(* CODESYS project festo_motion_fhpp_3.library
   Company: Festo AG & Co. KG
   DefaultNamespace: FML
   Title: Festo_Motion_FHPP_3
   Description: Library to control and parameterise drives from Festo with FHPP
   Author: chmm
   Version: 3.5.7.21

Project tree, tasks and I/O mapping:
  libraries: Standard, * (System)
  Enums/
    data type E_FML_DIAG_EVENT
    data type E_FML_FPC_MODUS
    data type E_FML_FPC_REQ_ID
    data type E_FML_FPC_RESP_ID
    data type E_FML_OPM
    data type E_FML_DEVICE_TYPE
    data type E_FML_FPC_STATUS_CATEGORY
    data type E_FML_FPC_STATUS_ID_FUNCTION_BLOCK
    data type E_FML_FPC_STATUS_ID_FILE_TRANSFER
  Internal/
    Blocks/
      ReadWriteData/
        function block FHPP_PLUS_Read [ST]
        function block FPC_Write [ST]
        function block FHPP_Read [ST]
        function block FHPP_PLUS_Write [ST]
        function block FHPP_Write [ST]
        function block FPC_Read [ST]
      FaultString/
        function ErrorList_CMMP_AS [ST]
        function ErrorList_CMMD_CMMS [ST]
        function ErrorList_CMMO_ST_EMCA_EC [ST]
        function FaultString [ST]
        function ErrorList_SFC_MTR [ST]
      function GetStatusMessage [ST]
      function GetStateOPMString [ST]
      function FML_DiagEventString [ST]
      function FML_TimeStamp [ST]
      function FormatInt [ST]
      function GetOPMString [ST]
    Enums/
      data type FML_FPC_FILE_TRANSFER_CONTROL
    Structs/
      FPC/
        data type DT_FPC
        data type DT_FPC_DATA
      FHPP/
        data type DT_CCON
        data type DT_CPOS
        data type DT_SCON
        data type DT_FHPP_DATA_IN
        data type DT_SPOS
        data type DT_FHPP
        data type DT_FHPP_DATA_OUT
      FHPP_PLUS/
        data type DT_FHPP_PLUS_OBJECT
        data type DT_FHPP_PLUS
      data type UCHAR
  Structs/
    data type DT_FML_REF
    data type DT_FML_PRM_DESCRIPTION
    data type DT_FML_PRM_DIAGMESSAGE
    data type DT_FML_DiagTable
    data type DT_FML_STATUS
    data type DT_FML_FPC_FILE_TRANSFER
  VISU/
    visualisation VIS_FPC_PNU
    visualisation VIS_FPC_DIAG_BUFFER
    visualisation VIS_FPC_DIRMP
    visualisation VIS_FPC_DATA_OBJECT
    visualisation VIS_FHPP_CTRL
    visualisation VIS_FPC_DIAG
    visualisation VIS_FPC_MULTI
    visualisation VIS_FPC_FILE_ARRAY
  Blocks/
    function block FHPP_CTRL [ST]
    function block FML_Read [ST]
    function block FML_Write [ST]
    Parameterize/
      function block FPC_DIAG_BUFFER [ST]
      function block FPC_MULTI [ST]
      function block FPC_PNU [ST]
      function block FPC_DATA_OBJECT [ST]
      function block FPC_DIAG [ST]
      function block FPC_FILE_ARRAY [ST]: CalculateFilesize, NextSequence
      function block FPC_DIRMP [ST]
  text list GlobalTextList
*)

// Structs/DT_FML_REF
(* ============================================================================
   FESTO AG & Co. KG, Esslingen - Copyright 2013. All rights reserved.                       
 ---------------------------------------------------------------------
 Data Type:     DT_FML_REF  
 Description:   data structure for Parametertransmission
 Version:       V3.1        
 Composer:      bejk
 Last Update:   26.06.2014                                                                           
 ---------------------------------------------------------------------
DATE        Name              	Activity                                                                              
11.03.2009  Benjamin Kilgus   	V1.0: created
13.05.2013  Rudolf Schenke    	V3.0: Formatting only
01.04.2014	Benjamin Kilgus	  	V3.1: extended to funktionality of EFPC
26.06.2014	Benjamin Kilgus	  	V3.1: extended FPCC_Packet/ FPCS_Packet
22.06.2015	Christian Hammer	adaptation to use this FB for all drives
08.09.2015	Christian Hammer	deleted 'ErrStr' with Error information
============================================================================ *)

TYPE DT_FML_REF :
	STRUCT
		(*data*)
		FHPP				: DT_FHPP;					// FHPP data
		FPC					: DT_FPC;					// FPC data
		FHPP_PLUS			: DT_FHPP_PLUS;				// FHPP+ data
	
		(*adjustments*)
		Modbus				: BOOL;						// Modbus is using
		HighByteFirst		: BOOL;						// Byteorder
		FPC_active			: BOOL;						// ParameterChannel (FPC) in use
	  	DeviceType			: E_FML_DEVICE_TYPE;		// Type of the Controller
		
		(*component infos*)
		MemberID	    	: INT:= 0;					// Current Member-ID
	 	MemberIDmax			: INT:= 0; 					// Maximum Member-ID
	  	Done          		: BOOL;     				// Execution Done 
	  	Err           		: BOOL;     				// Fault occured   
		
		(*request*)
		PNU           		: INT;	     				// Number of the Parameter 
	  	Subindex      		: DINT;    					// Subindex of the Parameter to Exchange 
		Value  				: DINT;     				// Value of the Parameter to Exchange
		DatatypeWR      	: USINT;    				// Length of the Parameter to Exchange in Byte
		ReqID				: E_FML_FPC_REQ_ID;
		FPCC_Packet			: DT_FML_FPC_FILE_TRANSFER; // File Transfer Packet Control
		FPCC_Modus			: DINT; 	  				// modus of parameter channel control

		(*response*)
		ActPNU        		: INT;	     				// Actual Number of the Parameter
	  	ActSubindex   		: DINT;    					// Actual Subindex of the Parameter 
	  	ActValue  			: DINT;     				// Read Value of Parameter
		DatatypeRD      	: USINT;    				// Actual Length of the Parameter in Byte
	  	RespID				: E_FML_FPC_RESP_ID;
	  	FPCS_Packet			: DT_FML_FPC_FILE_TRANSFER; // File Transfer Packet Status
		FPCS_Modus			: DINT; 	  				// modus of parameter channel status 
  END_STRUCT
END_TYPE

// Structs/DT_FML_PRM_DESCRIPTION
(* ============================================================================
   FESTO AG & Co. KG, Esslingen - Copyright (c) 2015. All rights reserved.                                   								
  -----------------------------------------------------------------------------  
 Description:    data structure for discription of the parameter   
 Last Update:    25.06.2014                                                                           
 ------------------------------------------------------------------------------
 Date        Name              	Activity                                                                              
 25.06.2014	 Benjamin Kilgus	created
 
 ============================================================================ *)

TYPE DT_FML_PRM_DESCRIPTION :
  STRUCT
	  PNU      	: INT ;		(* parameter number *)
	  SUBINDEX 	: INT ;		(* subindex of parameter *)
	  ACCESS   	: INT ;		(* 0 = read parameter / 1 = write parameter*)
	  VALUE    	: DINT ;	(* parameter value*)
	  Length	: USINT;	(* length of the parameter to exchange in byte (only necessary for SFC-DC and MTR-DCI) *)
  END_STRUCT
END_TYPE

// Structs/DT_FML_PRM_DIAGMESSAGE
(* ============================================================================
   FESTO AG & Co. KG, Esslingen - Copyright (c) 2015. All rights reserved.                                   								
  -----------------------------------------------------------------------------  
 Description:    data structure for diagnosis message   
 Last Update:    25.06.2014                                                                           
 ------------------------------------------------------------------------------
 Date        Name              	Activity                                                                              
 25.06.2014	 Benjamin Kilgus	created
 ============================================================================ *)

TYPE DT_FML_PRM_DIAGMESSAGE :
  STRUCT
	  DiagEvent          :E_FML_DIAG_EVENT;   	// event of message PNU 200/ PNU 210
	  DiagMsgNumber      :DINT;   			 	// message number PNU 201/ PNU 211
	  DiagTimeStamp      :DWORD;  				// time stamp of message PNU 202/ PNU 212
	  DiagMsgDescription :STRING; 				// description of message
  END_STRUCT
END_TYPE

// Enums/E_FML_DIAG_EVENT
(* ============================================================================
   FESTO AG & Co. KG, Esslingen - Copyright (c) 2015. All rights reserved.                                   								
  -----------------------------------------------------------------------------  
 Description:    enumeration for FML diagnosis event of the motorcontroller  
 Last Update:    22.06.2015                                                                           
 ------------------------------------------------------------------------------
 Date        Name                Activity                                                                              
 08.04.2014  Benjamin Kilgus	 created	 
 ============================================================================ *)

TYPE E_FML_DIAG_EVENT :
(
	none 				:= 0,
	error_comes     	:= 1,
	error_gone			:= 2,
	error_quit			:= 3,
	overflow_timestamp	:= 4,
	warning_comes		:= 5,
	warning_gone		:= 6,
	start_up_event  	:= 7,
	configuration		:= 8,
	information			:= 9
)INT;
END_TYPE

// Enums/E_FML_FPC_MODUS
(* ============================================================================
   FESTO AG & Co. KG, Esslingen - Copyright (c) 2015. All rights reserved.                                   								
  -----------------------------------------------------------------------------  
 Description:    enumeration for FML FPC Modus   
 Last Update:    25.06.2014                                                                           
 ------------------------------------------------------------------------------
 Date        Name              	Activity                                                                              
 01.04.2014  Benjamin Kilgus   	created 
 25.06.2014	Benjamin Kilgus	   	Type 4 and 5 added
 ============================================================================ *)

TYPE E_FML_FPC_MODUS :
(
	FML_FPC_MODUS_PNU_11BIT 	    := 0,	// transmit PNU 11 bit
	FML_FPC_MODUS_PNU_16BIT	 	    := 1,	// transmit PNU 16 bit
	FML_FPC_MODUS_DATA_OBJECT		:= 2,	// transmit internal data object
	FML_FPC_MODUS_CAN				:= 3,	// transmit CAN object
	FML_FPC_MODUS_ParameterFile	  	:= 4,	// transmit parameter file
	FML_FPC_MODUS_FirmwareUpdate  	:= 5	// transmit firmware file
)INT;
END_TYPE

// Enums/E_FML_FPC_REQ_ID
(* ============================================================================
   FESTO AG & Co. KG, Esslingen - Copyright (c) 2015. All rights reserved.                                   								
  -----------------------------------------------------------------------------  
 Description:    enumeration for FML FPC Modus   
 Last Update:    25.06.2014                                                                           
 ------------------------------------------------------------------------------
 Date        Name                Activity                                                                              
 25.06.2014	Benjamin Kilgus		 created
 ============================================================================ *)

TYPE E_FML_FPC_REQ_ID :
(
	FML_FPC_REQ_none	 			:= 0,	
	FML_FPC_REQ_read		 		:= 1,	
	FML_FPC_REQ_write_word			:= 2,	
	FML_FPC_REQ_write_dword			:= 3,	
	FML_FPC_REQ_read_file			:= 4,	
	FML_FPC_REQ_write_file			:= 5,
	FML_FPC_REQ_read_array			:= 6,
	FML_FPC_REQ_write_array_word	:= 7,
	FML_FPC_REQ_write_array_dword	:= 8,
	FML_FPC_REQ_read_array_elements	:= 9,
	FML_FPC_REQ_reseved0			:= 10,
	FML_FPC_REQ_write_byte			:= 11,
	FML_FPC_REQ_write_array_byte	:= 12,
	FML_FPC_REQ_read_lower_limit	:= 13,
	FML_FPC_REQ_read_upper_limit	:= 14	
)INT;
END_TYPE

// Enums/E_FML_FPC_RESP_ID
(* ============================================================================
   FESTO AG & Co. KG, Esslingen - Copyright (c) 2015. All rights reserved.                                   								
  -----------------------------------------------------------------------------  
 Description:    enumeration for FML FPC Modus   
 Last Update:    25.06.2014                                                                           
 ------------------------------------------------------------------------------
 Date        Name                Activity                                                                              
 25.06.2014	Benjamin Kilgus		 created
 ============================================================================ *)

TYPE E_FML_FPC_RESP_ID :
(
	FML_FPC_RESP_none	 				:= 0,	
	FML_FPC_RESP_word_done	 			:= 1,	
	FML_FPC_RESP_dword_done				:= 2,	
	FML_FPC_RESP_file_done				:= 3,	
	FML_FPC_RESP_word_array_done		:= 4,	
	FML_FPC_RESP_dword_array_done		:= 5,
	FML_FPC_RESP_error					:= 7,
	FML_FPC_RESP_read_array_elements	:= 9,
	FML_FPC_RESP_reseved0				:= 10,
	FML_FPC_RESP_byte_done				:= 11,
	FML_FPC_RESP_byte_array_done		:= 12		
)INT;
END_TYPE

// Enums/E_FML_OPM
(* ============================================================================
   FESTO AG & Co. KG, Esslingen - Copyright (c) 2015. All rights reserved.                                   								
  -----------------------------------------------------------------------------  
 Description:    enumeration for FML OPM   
 Last Update:    25.06.2014                                                                           
 ------------------------------------------------------------------------------
 Date        Name                Activity                                                                              
 25.06.2014	Benjamin Kilgus		 created
 ============================================================================ *)

TYPE E_FML_OPM :(
	OPM_RECORD_SEL	:= 0,
	OPM_DIRECT_POS	:= 1,
	OPM_DIRECT_TRQ	:= 5,
	OPM_DIRECT_VELO := 9
)INT;
END_TYPE

// Enums/E_FML_DEVICE_TYPE
(* ============================================================================
   FESTO AG & Co. KG, Esslingen - Copyright (c) 2015. All rights reserved.                                   								
  -----------------------------------------------------------------------------  
 Description:    enumeration for FML device type for different motorcontroller  
 Last Update:    13.11.2017                                                                           
 ------------------------------------------------------------------------------
 Date        Name               Activity                                                                              
 22.06.2015	Christian Hammer	created
 13.11.2017	Christian Hammer	added SFC-DC and MTR-DCI controller 
 ============================================================================ *)

TYPE E_FML_DEVICE_TYPE :(
  CMMO_ST	:= 10,
  EMCA_EC	:= 20,
  CMMP_AS	:= 30, 
  CMMS_AS	:= 40,
  CMMS_ST   := 50,
  CMMD_AS	:= 60,
  SFC_DC	:= 70,
  MTR_DCI	:= 80
)INT;
END_TYPE

// Enums/E_FML_FPC_STATUS_CATEGORY
(* ============================================================================
   FESTO AG & Co. KG, Esslingen - Copyright (c) 2015. All rights reserved.                                   								
  -----------------------------------------------------------------------------  
 Description:    enumeration for FML error categories  
 Last Update:    22.06.2015                                                                           
 ------------------------------------------------------------------------------
 Date      		Name              		Activity                                                                              
 08.04.2014  	Benjamin Kilgus	 		created
 08.09.2015	 	Christian Hammer		deleted cat filesystem	 
 ============================================================================ *)

TYPE E_FML_FPC_STATUS_CATEGORY :
(
	FML_no_category			:= 0,
	FML_function_block		:= 1,
	FML_reserved			:= 2,
	FML_parameter_transfer	:= 3	
)DINT;
END_TYPE

// Enums/E_FML_FPC_STATUS_ID_FUNCTION_BLOCK
(* ============================================================================
   FESTO AG & Co. KG, Esslingen - Copyright (c) 2015. All rights reserved.                                   								
  -----------------------------------------------------------------------------  
 Description:    enumeration for FML status ID of function blocks 
 Last Update:    22.06.2015                                                                           
 ------------------------------------------------------------------------------
 Date        	Name               		Activity                                                                              
 08.04.2014  	Benjamin Kilgus	 		created
 08.09.2015	 	Christian Hammer		changed name of enum		 
 ============================================================================ *)

TYPE E_FML_FPC_STATUS_ID_FUNCTION_BLOCK :
(
	FML_no_error						:= 0, 		// finished with no error
	FML_init_active						:= 1, 		// init of function block is active
	FML_fb_busy							:= 2, 		// transfer is active/busy
	FML_other_fb_active					:= 10, 		// execution not possible because another FB is active
	FML_fb_timeout						:= 20,		// timeout of the function block (no response from the controller)
	FML_wrong_device					:= 30,		// execution not possible for this device type
	FML_wrong_access_value				:= 40,   	// wrong value for ACCESS in function block 'FPC_MULTI'
	FML_pointer_to_zero					:= 50, 		// no input on either SizeOf or address of parameter
	FML_pointer_wrong_size				:= 51, 		// wrong size of parameter size has to by n*Size of DT_FML_PRM_DESCRIPTION
	FML_fhpp_plus_value_not_valid		:= 60		// wrong value for FHPP+ data mapping in function block 'FML_Read' or 'FML_Write'
)INT;
END_TYPE

// Enums/E_FML_FPC_STATUS_ID_FILE_TRANSFER
(* ============================================================================
   FESTO AG & Co. KG, Esslingen - Copyright (c) 2015. All rights reserved.                                   								
  -----------------------------------------------------------------------------  
 Description:    enumeration for FML status ID for file transfer   
 Last Update:    22.06.2015                                                                           
 ------------------------------------------------------------------------------
 Date        	Name               		Activity                                                                              
 08.04.2014  	Benjamin Kilgus	 		created
 08.09.2015	 	Christian Hammer		deleted changed name of enum 
 08.09.2015	 	Christian Hammer		set offset of 1000			 
 ============================================================================ *)

TYPE E_FML_FPC_STATUS_ID_FILE_TRANSFER :
(
	FML_no_file_err		:= 1000,
	FML_wrong_sequ		:= 1001,
	FML_time_out_pack	:= 1002,
	FML_wrong_pack		:= 1003,
	FML_false_instr		:= 1004,
	FML_read_err		:= 1005,
	FML_write_err		:= 1006,
	FML_volume_err		:= 1007,
	FML_par_file_err	:= 1008,
	FML_fault_receipt	:= 1009,
	FML_time_out		:= 1010,
	FML_err_at_open		:= 1011,
	FML_err_at_close	:= 1012,
	FML_err_at_delete	:= 1013,
	FML_err_at_create 	:= 1014,
	FML_not_exist		:= 1015,
	FML_err_at_read		:= 1016,
	FML_not_used		:= 1017,
	FML_err_at_write	:= 1018,
	FML_direction_err	:= 1019,
	FML_file_name_err	:= 1020,
	FML_size_err		:= 1021,
	FML_incomplete		:= 1022
) DINT;
END_TYPE

// Internal/Enums/FML_FPC_FILE_TRANSFER_CONTROL
(* ============================================================================
   FESTO AG & Co. KG, Esslingen - Copyright (c) 2015. All rights reserved.                                   								
  -----------------------------------------------------------------------------  
 Description:    data structure for file transfer control   
 Last Update:    25.06.2014                                                                           
 ------------------------------------------------------------------------------
 Date        Name              	Activity                                                                              
 25.06.2014	 Benjamin Kilgus	created
 ============================================================================ *)

TYPE FML_FPC_FILE_TRANSFER_CONTROL :
(
	FML_FPC_FILE_TRANSFER_active 	:= 0,	// exchange active
	FML_FPC_FILE_TRANSFER_start	 	:= 1,	// start exchange
	FML_FPC_FILE_TRANSFER_stop 		:= 2,	// stop exchange
	FML_FPC_FILE_TRANSFER_error 	:= 3,	// exchange error
	FML_FPC_FILE_TRANSFER_reserved	:= 4	

)USINT;
END_TYPE

// Internal/Structs/FPC/DT_FPC
(* ============================================================================
   FESTO AG & Co. KG, Esslingen - Copyright (c) 2015. All rights reserved.                                   								
  -----------------------------------------------------------------------------  
 Description:    data structure for FPC data 
 Last Update:    22.06.2015                                                                           
 ------------------------------------------------------------------------------
 Date        Name              	Activity                                                                              
 22.06.2015	 Christian Hammer	created
 ============================================================================ *)

TYPE DT_FPC :
	STRUCT
		IN  	: DT_FPC_DATA;
		OUT 	: DT_FPC_DATA;
	END_STRUCT
END_TYPE

// Internal/Structs/FPC/DT_FPC_DATA
(* ============================================================================
   FESTO AG & Co. KG, Esslingen - Copyright (c) 2015. All rights reserved.                                   								
  -----------------------------------------------------------------------------  
 Description:    data structure for FPC input and output data   
 Last Update:    22.06.2015                                                                           
 ------------------------------------------------------------------------------
 Date        Name              	Activity                                                                              
 22.06.2015	 Christian Hammer	created
 ============================================================================ *)

TYPE DT_FPC_DATA :
	STRUCT
		ModeAK 		: BYTE;
		IND 		: BYTE;
		ParID		: INT;
		Value 		: DINT;
	END_STRUCT
END_TYPE

// Internal/Structs/FHPP/DT_CCON
(* ============================================================================
   FESTO AG & Co. KG, Esslingen - Copyright (c) 2015. All rights reserved.                                   								
  -----------------------------------------------------------------------------  
 Description:    structure for CCON data (control byte 1)   
 Last Update:    22.06.2015                                                                           
 ------------------------------------------------------------------------------
 Date        Name              	Activity                                                                              
 22.06.2015	 Christian Hammer	created
 ============================================================================ *)

TYPE DT_CCON :
	STRUCT
		ENABLE 	: BIT;
		STOP 	: BIT;
		BRAKE 	: BIT;
		RESET 	: BIT;
		res 	: BIT;
		LOCK 	: BIT;
		OPM1 	: BIT;
		OPM2 	: BIT;	
	END_STRUCT
END_TYPE

// Internal/Structs/FHPP/DT_CPOS
(* ============================================================================
   FESTO AG & Co. KG, Esslingen - Copyright (c) 2015. All rights reserved.                                   								
  -----------------------------------------------------------------------------  
 Description:    structure for CPOS data (control byte 2)   
 Last Update:    22.06.2015                                                                           
 ------------------------------------------------------------------------------
 Date        Name              	Activity                                                                              
 22.06.2015	 Christian Hammer	created
 ============================================================================ *)

TYPE DT_CPOS :
	STRUCT
		HALT 	: BIT;
		START 	: BIT;
		HOM 	: BIT;
		JOGP 	: BIT;
		JOGN 	: BIT;
		TEACH 	: BIT;
		CLEAR 	: BIT;
		res 	: BIT;	
	END_STRUCT
END_TYPE

// Internal/Structs/FHPP/DT_SCON
(* ============================================================================
   FESTO AG & Co. KG, Esslingen - Copyright (c) 2015. All rights reserved.                                   								
  -----------------------------------------------------------------------------  
 Description:    data structure for SCON data (status byte 1)   
 Last Update:    22.06.2015                                                                           
 ------------------------------------------------------------------------------
 Date        Name              	Activity                                                                              
 22.06.2015	 Christian Hammer	created
 ============================================================================ *)

TYPE DT_SCON :
	STRUCT
		ENABLED	: BIT;
		OPEN 	: BIT;
		WARN 	: BIT;
		FAULT 	: BIT;
		VLOAD 	: BIT;	
		FCT 	: BIT;
		OPM1 	: BIT;
		OPM2 	: BIT;	
	END_STRUCT
END_TYPE

// Internal/Structs/FHPP/DT_FHPP_DATA_IN
(* ============================================================================
   FESTO AG & Co. KG, Esslingen - Copyright (c) 2015. All rights reserved.                                   								
  -----------------------------------------------------------------------------  
 Description:    structure for FHPP input data 
 Last Update:    22.06.2015                                                                           
 ------------------------------------------------------------------------------
 Date        Name              	Activity                                                                              
 22.06.2015	 Christian Hammer	created
 29.02.2016	 Christian Hammer	changed type of ActValue1 from BYTE into SINT
 ============================================================================ *)

TYPE DT_FHPP_DATA_IN :
	STRUCT
		SCON 		: DT_SCON;
		SPOS 		: DT_SPOS;
		Byte3		: BYTE;
		ActValue1 	: SINT;
		ActValue2 	: DWORD;
	END_STRUCT
END_TYPE

// Internal/Structs/FHPP/DT_SPOS
(* ============================================================================
   FESTO AG & Co. KG, Esslingen - Copyright (c) 2015. All rights reserved.                                   								
  -----------------------------------------------------------------------------  
 Description:    data structure for SPOS data (status byte 2)   
 Last Update:    22.06.2015                                                                           
 ------------------------------------------------------------------------------
 Date        Name              	Activity                                                                              
 22.06.2015	 Christian Hammer	created
 ============================================================================ *)

TYPE DT_SPOS :
	STRUCT
		HALT 	: BIT;
		ACK 	: BIT;
		MC 		: BIT;
		TEACH 	: BIT;
		MOV 	: BIT;
		DEV 	: BIT;
		STILL 	: BIT;
		REF 	: BIT;	
	END_STRUCT
END_TYPE

// Internal/Structs/FHPP/DT_FHPP
(* ============================================================================
   FESTO AG & Co. KG, Esslingen - Copyright (c) 2015. All rights reserved.                                   								
  -----------------------------------------------------------------------------  
 Description:    data structure for FHPP data   
 Last Update:    22.06.2015                                                                           
 ------------------------------------------------------------------------------
 Date        Name              	Activity                                                                              
 22.06.2015	 Christian Hammer	created
 ============================================================================ *)

TYPE DT_FHPP :
	STRUCT
		IN  	: DT_FHPP_DATA_IN;
		OUT 	: DT_FHPP_DATA_OUT;
	END_STRUCT
END_TYPE

// Internal/Structs/FHPP/DT_FHPP_DATA_OUT
(* ============================================================================
   FESTO AG & Co. KG, Esslingen - Copyright (c) 2015. All rights reserved.                                   								
  -----------------------------------------------------------------------------  
 Description:    data structure for FHPP output data 
 Last Update:    22.06.2015                                                                           
 ------------------------------------------------------------------------------
 Date        Name              	Activity                                                                              
 22.06.2015	 Christian Hammer	created
 ============================================================================ *)

TYPE DT_FHPP_DATA_OUT :
	STRUCT
		CCON 		: DT_CCON;
		CPOS 		: DT_CPOS;
		Byte3 		: BYTE;
		SetValue1 	: BYTE;
		SetValue2 	: DWORD;
	END_STRUCT
END_TYPE

// Structs/DT_FML_DiagTable
(* ============================================================================
   FESTO AG & Co. KG, Esslingen - Copyright (c) 2015. All rights reserved.                                   								
  -----------------------------------------------------------------------------  
 Description:    data structure for diagnosis visualisation   
 Last Update:    25.06.2014                                                                           
 ------------------------------------------------------------------------------
 Date        Name              	Activity                                                                              
 25.06.2014	 Benjamin Kilgus	created
 ============================================================================ *)

TYPE DT_FML_DiagTable :
  STRUCT
    sEvent    : STRING;
    sStamp    : STRING;
    sFault    : STRING;
    sText     : STRING;
  END_STRUCT
END_TYPE

// Structs/DT_FML_STATUS
(* ============================================================================
   FESTO AG & Co. KG, Esslingen - Copyright (c) 2015. All rights reserved.                                   								
  -----------------------------------------------------------------------------  
 Description:    data structure for Status output of the function blocks   
 Last Update:    25.06.2014                                                                           
 ------------------------------------------------------------------------------
 Date        Name              	Activity                                                                              
 08.09.2015	Christian Hammer	created
 ============================================================================ *)

TYPE DT_FML_STATUS:
  STRUCT
	  Err 		: BOOL;			// error bit
	  Cat		: DINT;			// status category
	  ID		: DINT;			// status ID
	  Msg		: STRING;	 	// status message 
  END_STRUCT
END_TYPE

// Internal/Structs/FHPP_PLUS/DT_FHPP_PLUS_OBJECT
(* ============================================================================
   FESTO AG & Co. KG, Esslingen - Copyright (c) 2015. All rights reserved.                                   								
  -----------------------------------------------------------------------------  
 Description:    structure for FHPP+ objects   
 Last Update:    19.08.2015                                                                           
 ------------------------------------------------------------------------------
 Date        Name              	Activity                                                                              
 19.08.2015	 Christian Hammer	created
 ============================================================================ *)

TYPE DT_FHPP_PLUS_OBJECT :
	STRUCT
		Object1		: DINT;
		Object2		: DINT;
		Object3		: DINT;
		Object4		: DINT;
		Object5		: DINT;
		Object6		: DINT;
		Object7		: DINT;
		Object8		: DINT;
		Object9		: DINT;
		Object10	: DINT;
	END_STRUCT
END_TYPE

// Internal/Structs/FHPP_PLUS/DT_FHPP_PLUS
(* ============================================================================
   FESTO AG & Co. KG, Esslingen - Copyright (c) 2015. All rights reserved.                                   								
  -----------------------------------------------------------------------------  
 Description:    structure for FHPP+ data   
 Last Update:    19.08.2015                                                                           
 ------------------------------------------------------------------------------
 Date        Name              	Activity                                                                              
 19.08.2015	 Christian Hammer	created
 ============================================================================ *)

TYPE DT_FHPP_PLUS :
	STRUCT
		IN		: DT_FHPP_PLUS_OBJECT;
		OUT		: DT_FHPP_PLUS_OBJECT;
	END_STRUCT
END_TYPE

// Structs/DT_FML_FPC_FILE_TRANSFER
(* ============================================================================
   FESTO AG & Co. KG, Esslingen                                                    								
  -----------------------------------------------------  
 Description:    for FML_FPC_FILE_TRANSFER   
 Last Update:    25.06.2014                                                                           
 -----------------------------------------------------
Date        Name              Activity                                                                              
25.06.2014	Benjamin Kilgus		created
============================================================================ *)
TYPE DT_FML_FPC_FILE_TRANSFER :
	STRUCT
		Control		  		: INT;	
		BitSequenceNr 		: INT;
		Data			    : ARRAY[1..6] OF BYTE;
	END_STRUCT
END_TYPE;

// Internal/Structs/UCHAR
{library private}
// Union for hex formatting in function "Format"
TYPE UCHAR :
  UNION
    str  : STRING[1]; // String from Byte
    char : BYTE;      // Target for char calculation
  END_UNION
END_TYPE

// Internal/Blocks/ReadWriteData/FHPP_PLUS_Read
(* ===============================================================================
   FESTO AG & Co. KG, Esslingen - Copyright 2015. All rights reserved.                       
 ---------------------------------------------------------------------------------
 Functionblock:  FHPP_PLUS_Read  
 Description:    function block to read and mapp the FHPP+ data from the controller
 Version:        V 3.5.4.4        
 Composer:       chmm 
 Last Update:    19.08.2015                                                                           
------------------------------------------------------------------------------- *)
{library private}
(* ----------------------------------------------------------------------------
Date        Name            	Activity                                                                              
19.08.2015	Christian Hammer	created
=============================================================================== *)
{library public}

FUNCTION_BLOCK FHPP_PLUS_Read

VAR_IN_OUT
	FML_REF					: DT_FML_REF;						// structure of the parameter to control and parametrize the motorcontroller
END_VAR	

VAR_INPUT
	FHPP_PLUS_Source1		: ARRAY [0..7] OF BYTE;				// first 8 bytes of FHPP+ input data (from controller)
	FHPP_PLUS_Source2		: ARRAY [0..7] OF BYTE;				// second 8 bytes of FHPP+ input data (from controller)
	FHPP_PLUS_Source3		: ARRAY [0..7] OF BYTE;				// third 8 bytes of FHPP+ input data (from controller)
	PlcConfigFHPP_PLUS_IN	: UDINT;							// plc configuration code for the FHPP+ input(is displayed in the Festo Configuration Tool (FCT))
END_VAR

VAR_OUTPUT
	Status          		: DT_FML_STATUS;    				// return value of function block
END_VAR

VAR
	FHPP_PLUS_DATA_IN		: ARRAY[0..23] OF BYTE;				// intern variable to buffer the FHPP+ input data
	pDataArray				: POINTER TO ARRAY[0..7] OF BYTE;	// pointer to copy the FHPP+ data from the bus into the intern buffer variable - FHPP_PLUS_DATA_IN
	pFHPP_PLUS_Object		: POINTER TO ARRAY[0..9] OF DINT;	// pointer to copy the data from intern buffer variable to the FML_REF - FML_REF.FHPP_PLUS.IN
	stConfigFHPP_PLUS		: STRING[9];						// string with the plc configuration code for the FHPP+ input(is displayed in the Festo Configuration Tool (FCT))
	iCount					: INT;								// counter variable for the loop
	iAddress				: INT;								// counter variable for address of the pointer
	iObject					: INT;								// counter variable for FHPP+ objects in FML_REF
END_VAR

(***********************************************************************************************************************************************
*********** INPUT FHPP+ DATA *******************************************************************************************************************
***********************************************************************************************************************************************)

Status.Err:=FALSE; Status.Cat:=FML_function_block; Status.ID:=FML_init_active;

// inizialize the variables
iAddress			:= 0;
iObject				:= 0;
iCount				:= 0;

// inizialize the pointer to FML_REF
pFHPP_PLUS_Object	:= ADR(FML_REF.FHPP_PLUS.IN);

// change PLC-Config from FCT (is a INT) into a string
stConfigFHPP_PLUS	:= UDINT_TO_STRING(PlcConfigFHPP_PLUS_IN);

Status.Err:=FALSE; Status.Cat:=FML_function_block; Status.ID:=FML_fb_busy;

// write input data from the bus into FHPP_PLUS_DATA_IN
IF FML_REF.Modbus THEN											// Modbus word swapping
	FHPP_PLUS_DATA_IN[0]	:= FHPP_PLUS_Source1[1];
	FHPP_PLUS_DATA_IN[1]	:= FHPP_PLUS_Source1[0];
	FHPP_PLUS_DATA_IN[2]	:= FHPP_PLUS_Source1[3];
	FHPP_PLUS_DATA_IN[3]	:= FHPP_PLUS_Source1[2];
	FHPP_PLUS_DATA_IN[4]	:= FHPP_PLUS_Source1[5];
	FHPP_PLUS_DATA_IN[5]	:= FHPP_PLUS_Source1[4];
	FHPP_PLUS_DATA_IN[6]	:= FHPP_PLUS_Source1[7];
	FHPP_PLUS_DATA_IN[7]	:= FHPP_PLUS_Source1[6];
	FHPP_PLUS_DATA_IN[8]	:= FHPP_PLUS_Source2[1];
	FHPP_PLUS_DATA_IN[9]	:= FHPP_PLUS_Source2[0];
	FHPP_PLUS_DATA_IN[10]	:= FHPP_PLUS_Source2[3];
	FHPP_PLUS_DATA_IN[11]	:= FHPP_PLUS_Source2[2];
	FHPP_PLUS_DATA_IN[12]	:= FHPP_PLUS_Source2[5];
	FHPP_PLUS_DATA_IN[13]	:= FHPP_PLUS_Source2[4];
	FHPP_PLUS_DATA_IN[14]	:= FHPP_PLUS_Source2[7];
	FHPP_PLUS_DATA_IN[15]	:= FHPP_PLUS_Source2[6];
	FHPP_PLUS_DATA_IN[16]	:= FHPP_PLUS_Source3[1];
	FHPP_PLUS_DATA_IN[17]	:= FHPP_PLUS_Source3[0];
	FHPP_PLUS_DATA_IN[18]	:= FHPP_PLUS_Source3[3];
	FHPP_PLUS_DATA_IN[19]	:= FHPP_PLUS_Source3[2];
	FHPP_PLUS_DATA_IN[20]	:= FHPP_PLUS_Source3[5];
	FHPP_PLUS_DATA_IN[21]	:= FHPP_PLUS_Source3[4];
	FHPP_PLUS_DATA_IN[22]	:= FHPP_PLUS_Source3[7];
	FHPP_PLUS_DATA_IN[23]	:= FHPP_PLUS_Source3[6];
		
ELSE															// normal fieldbus: copy only
	pDataArray		:= ADR(FHPP_PLUS_DATA_IN[0]);
	pDataArray^		:= FHPP_PLUS_Source1;
	pDataArray		:= ADR(FHPP_PLUS_DATA_IN[8]);
	pDataArray^		:= FHPP_PLUS_Source2;
	pDataArray		:= ADR(FHPP_PLUS_DATA_IN[16]);
	pDataArray^		:= FHPP_PLUS_Source3;
END_IF


// FOR loop to copy input data from the bus into the intern FHPP+ objects 
FOR (iCount := 0) TO 9 BY 1 DO

	// read the PLC-Config string from FCT to copy the right number of bytes into the intern FHPP+ object
	CASE stConfigFHPP_PLUS[iCount] OF
		
		49:	//ascii code for '1'	--> the size of the object is 8 BITs --> copy one BYTE into the FHPP+ object
			pFHPP_PLUS_Object^[iObject]		:= (FHPP_PLUS_DATA_IN[iAddress]);
			iAddress						:= iAddress + 1;		// increment the counter variable for address of the pointer in increments of 1
			
			
		50:	//ascii code for '2'	--> the size of the object is 16 BITs --> copy two BYTEs into the FHPP+ object
			IF FML_REF.HighByteFirst THEN	// byteorder = high byte first 
				pFHPP_PLUS_Object^[iObject]	:= (FHPP_PLUS_DATA_IN[iAddress+1] + FHPP_PLUS_DATA_IN[iAddress]*256);		
				
			ELSE							// byteorder = low byte first 
				pFHPP_PLUS_Object^[iObject]	:= (FHPP_PLUS_DATA_IN[iAddress] + FHPP_PLUS_DATA_IN[iAddress+1]*256);		
			END_IF
			iAddress						:= iAddress + 2;		// increment the counter variable for address of the pointer  in increments of 2
		
			
		52:	//ascii code for '4'	--> the size of the object is 32 BITs --> copy four BYTEs into the FHPP+ object
			IF FML_REF.HighByteFirst THEN	// byteorder = high byte first
				pFHPP_PLUS_Object^[iObject]	:= UDINT_TO_DINT(FHPP_PLUS_DATA_IN[iAddress+3] + FHPP_PLUS_DATA_IN[iAddress+2]*256 + FHPP_PLUS_DATA_IN[iAddress+1]*65536 + FHPP_PLUS_DATA_IN[iAddress]*16777216);	
	
			ELSE							// byteorder = low byte first	
				pFHPP_PLUS_Object^[iObject]	:= UDINT_TO_DINT(FHPP_PLUS_DATA_IN[iAddress] + FHPP_PLUS_DATA_IN[iAddress+1]*256 + FHPP_PLUS_DATA_IN[iAddress+2]*65536 + FHPP_PLUS_DATA_IN[iAddress+3]*16777216);		
			END_IF
			iAddress						:= iAddress + 4;		// increment the counter variable for address of the pointer in increments of 4
			
		
		48, 51, 53, 54, 55, 56, 57:	//ascii code for '0', '3', '5', '6', '7', '8', '9' --> wrong number is in the plc configuration code for the FHPP+ input(is displayed in the Festo Configuration Tool (FCT))
			Status.Err:=TRUE; Status.Cat:=FML_function_block; Status.ID:=FML_fhpp_plus_value_not_valid;
			RETURN;
			
		ELSE // else fill up the remaining objects with zero	
			pFHPP_PLUS_Object^[iObject]		:= 0;	
		
	END_CASE
	
	iObject									:= iObject + 1;			// increment the counter variable for FHPP+ objects in FML_REF

END_FOR

Status.Err:=FALSE; Status.Cat:=FML_no_category; Status.ID:=FML_no_error;

(* ===== end of function block ============================= *)

END_FUNCTION_BLOCK

// Blocks/Parameterize/FPC_DIAG_BUFFER
(* ============================================================================
   FESTO AG & Co. KG, Esslingen - Copyright 2015. All rights reserved.                       
 -----------------------------------------------------
 Functionblock:  FPC_DIAG_BUFFER
 Description:    fuction block to read diagnostic buffer
 Version:        V3.5.7.21         
 Composer:       bejk 
 Last Update:    13.11.2017                                                                           
------------------------------------------------------------------------------- *)
{library private}
(* ----------------------------------------------------------------------------
Date        Name              	Activity                                                                              
10.04.2014  Benjamin Kilgus   	created from MTR_DCI_PRM_DIAG
14.09.2014	Rudolf Schenke		Missing FML_REF.ReqID added
								VISU correction (Timestamp, Message 0xnn) 
09.02.2015  Rudolf Schenke    	implement 16-bit mode with hide preset
22.06.2015	Christian Hammer	adaptation to use this FB for all drives
04.09.2015  Christian Hammer	error handling (deleted RETVAL, created Status)
13.11.2017	Christian Hammer	added SFC-DC and MTR-DCI controller (add step 18 and 19)
============================================================================ *)
{library public}

(* use this function block only with the function blocks FML_Read and FML_Write *)

FUNCTION_BLOCK FPC_DIAG_BUFFER

VAR_IN_OUT
	FML_REF        		: DT_FML_REF;								// structure of the parameter to control and parametrize the motorcontroller
END_VAR

VAR_INPUT															
	Execute         	: BOOL;  									// perfrom data exchange
END_VAR

VAR_OUTPUT
	Done        		: BOOL;										// transmission done	
	Error				: BOOL; 									// transmission fault
	Status				: DT_FML_STATUS;							// structure with the status information of the function block and FPC
	ValidEntries		: INT;										// amount of valid entries in buffer
	ParamNo     		: INT;										// no of current parameter
	DiagBuff    		: ARRAY [1..200] OF DT_FML_PRM_DIAGMESSAGE; // buffer with the diagnosis messages
END_VAR

{library private}

VAR
	bInit       		: BOOL	:=FALSE;							// status of inizialisation of the FB
	lMemberID   		: INT;										// local member ID of the FB								
	Step        		: INT;										// local step number
	awPNU       		: ARRAY [0..2] OF INT := [200, 201, 202];	// PNUs with the diagnosis informations
	ixPNU       		: INT;        								// index in awPNU
	diValue     		: DINT;       								// save read results  
	iSI         		: INT;      								// subindex
 	max_iSI				: INT;										// max number of the diagnosis messages (depends on drive)
	astVisu     		: ARRAY [1..200] OF DT_FML_DiagTable;		// buffer for FB visualization
	sEventBuffer		: STRING;									// description of the diagnose message
	
	TONInst				: TON;										// timer instance to monitor a timeout of the function block
	TimeStart			: BOOL;										// variable to start the timer instance
	TimeoutTime			: TIME := T#3S;								// timeout time
	
	TimerFwBug			: TON;										// timer because of FW bug in SFC-Dc and MTR-DCI
	StartTimerFwBug		: BOOL;										// variable to start TimerFwBug
END_VAR

VAR CONSTANT
	maxDiagBuffElements	: INT := 200;								// max number of diagnosis messages (CMMO and EMCA)
END_VAR

{library public}

(* ====== initial block routine ===================================== *)
(* ----- get MemberID for this function block ----------------------- *)
IF NOT bInit THEN 
 	FML_REF.MemberIDmax		:= FML_REF.MemberIDmax +1;
	lMemberID				:= FML_REF.MemberIDmax;
	bInit					:= TRUE;
	Status.Err:=FALSE; Status.Cat:=FML_function_block; Status.ID:=FML_init_active;
END_IF


(* ====== supervision of timeout ==================================== *)
(* ----- timer to monitor a timeout of the function block ------------*)
TimerFwBug(IN:= StartTimerFwBug, PT:= T#250MS);
TONInst(IN := TimeStart, PT := TimeoutTime);
IF TONInst.Q THEN
	Status.Err:=TRUE; Status.Cat:=FML_function_block; Status.ID:=FML_fb_timeout;
	Done					:= TRUE;
	Step					:= 100;
END_IF	


(* ===== logic part ================================================= *)
(* ----- ASSIGNMENT OF STATUS --------------------------------------- *)
IF NOT Execute AND(Step <> 0) THEN
	FML_REF.MemberID		:= 0;
	FML_REF.ReqID			:= FML_FPC_REQ_none;
	FML_REF.PNU				:= 0;
	FML_REF.Subindex		:= 0;
	FML_REF.Value			:= 0;
	Step					:= 0;
END_IF;

CASE Step OF
	0:(* init some variables *)
		Done					:= FALSE;
		TimeStart				:= FALSE;
		StartTimerFwBug			:= FALSE;
		ValidEntries			:= 0;
		ParamNo					:= 0;
		ixPNU					:= 0;    					// PNU array index
		Status.Err:=FALSE; Status.Cat:=FML_no_category; Status.ID:=FML_no_error;
	
		IF (FML_REF.MemberID = 0) AND Execute THEN
			FML_REF.MemberID		:= lMemberID;
			iSI						:= 1;    					// Subindex (counter)
			Step   					:= 10;						// read message
			Status.Err:=FALSE; Status.Cat:=FML_function_block; Status.ID:=FML_fb_busy;
			
		ELSIF (FML_REF.MemberID <> lMemberId) AND Execute THEN
			Status.Err:=FALSE; Status.Cat:=FML_function_block; Status.ID:=FML_other_fb_active;
		END_IF

	10:(* set size of the error memory  *)
		TimeStart					:= TRUE;
		IF NOT FML_REF.Done THEN
			TimeStart				:= FALSE;
			IF (FML_REF.DeviceType = CMMP_AS) THEN																			(*******CMMP-AS*******)	
				FML_REF.FPCC_Modus 	:= E_FML_FPC_MODUS.FML_FPC_MODUS_PNU_11BIT;
				max_iSI				:= 32;						// size of error memory = 32
				Step				:= 20;						
			ELSIF (FML_REF.DeviceType = CMMS_AS) OR (FML_REF.DeviceType = CMMS_ST) OR (FML_REF.DeviceType = CMMD_AS) THEN	(* CMMS_AS or CMMS_ST or CMMD_AS *)
				FML_REF.FPCC_Modus 	:= E_FML_FPC_MODUS.FML_FPC_MODUS_PNU_11BIT;
				max_iSI				:= 4;						// size of error memory = 4 
				Step				:= 20;	
			ELSIF (FML_REF.DeviceType = SFC_DC) OR (FML_REF.DeviceType = MTR_DCI) THEN										(* SFC-DC or MTR-DCI *)
				FML_REF.FPCC_Modus 	:= E_FML_FPC_MODUS.FML_FPC_MODUS_PNU_11BIT;
				max_iSI				:= 16;						// size of error memory = 16 
				Step				:= 20;		
			ELSE 																											(*******EMCA-EC or CMMO-ST*******)	
				FML_REF.FPCC_Modus 	:= E_FML_FPC_MODUS.FML_FPC_MODUS_PNU_16BIT;
				FML_REF.PNU			:= 204; 					// read PNU and Subindex with the number of valid entries
				FML_REF.Subindex	:= 4;   					
				Step				:= 12;
				FML_REF.ReqID		:= FML_FPC_REQ_read_array;
			END_IF	
		END_IF
  
	12:(* set number of the valid entries in the error memory (EMCA and CMMO) *)
		TimeStart					:= TRUE;
		IF FML_REF.Done AND NOT FML_REF.Err THEN
			TimeStart				:= FALSE;
			FML_REF.ReqID			:= FML_FPC_REQ_none;
			ValidEntries			:= DINT_TO_INT(FML_REF.ActValue);
			max_iSI					:= ValidEntries;			// size of error memory = ValidEntries (maximum = 200)
			Step					:= 20;
		ELSIF FML_REF.Done AND FML_REF.Err THEN
			Status.Err:=TRUE; Status.Cat:=FML_parameter_transfer; Status.ID:=FML_REF.ActValue;
			Step					:= 30;
		END_IF;  
		
  	18:	(* delay state because of FW bug from SFC-DC and MTR-DCI *)
		StartTimerFwBug				:= TRUE;	
		IF TimerFwBug.Q THEN
			StartTimerFwBug			:= FALSE;
			step 					:= 20;
		END_IF
		
	19:	(* delay state because of FW bug from SFC-DC and MTR-DCI *)
		StartTimerFwBug				:= TRUE;	
		IF TimerFwBug.Q THEN
			StartTimerFwBug			:= FALSE;
			step 					:= 21;
		END_IF	
	
	20: (* read error memory *)
		TimeStart					:= TRUE;
		IF NOT FML_REF.Done THEN
			TimeStart				:= FALSE;
			FML_REF.PNU				:= awPNU[ixPNU]; 			// PNUs with the diagnosis informations (200, 201, 202)
			FML_REF.Subindex		:= iSI;         			// subindex with the error number
			FML_REF.ReqID			:= FML_FPC_REQ_read_array;
			
			IF FML_REF.DeviceType = SFC_DC OR FML_REF.DeviceType = MTR_DCI THEN													(* SFC-DC or MTR-DCI *)
				Step				:= 19;
			ELSE																												(* CMMP-AS or CMMS-AS or CMMS-ST or EMCA-EC or CMMO-ST *)
				Step				:= 21;	
			END_IF
		END_IF;
				
	21:(* prepare next PNU *)
		TimeStart					:= TRUE;
		IF FML_REF.Done AND NOT FML_REF.Err THEN
			TimeStart				:= FALSE;
			FML_REF.ReqID			:= FML_FPC_REQ_none;
			FML_REF.PNU				:= 0;
			FML_REF.Subindex		:= 0;
			diValue					:= FML_REF.ActValue;
			CASE ixPNU OF
				0: // PNU for kind of event
				DiagBuff[iSI].DiagEvent				:= DINT_TO_INT(diValue);
				sEventBuffer						:= FML_DiagEventString(DINT_TO_DWORD(diValue));
	
				1: // PNU for diagnosis number
				DiagBuff[iSI].DiagMsgNumber			:= diValue;
				DiagBuff[iSI].DiagMsgDescription	:= FaultString(diValue, FML_REF.DeviceType);
			 
				2: // PNU for time stamp
				DiagBuff[iSI].DiagTimeStamp 		:= DINT_TO_DWORD(diValue);
				IF diValue <> 0 THEN
					astVisu[iSI].sEvent				:= sEventBuffer;
					astVisu[iSI].sStamp				:= FML_TimeStamp(DiagBuff[iSI].DiagTimeStamp,0);
					astVisu[iSI].sFault 			:= CONCAT('0x', FormatInt(DINT_TO_UDINT(DiagBuff[iSI].DiagMsgNumber),'%x2'));
					astVisu[iSI].sText  			:= DiagBuff[iSI].DiagMsgDescription;
					ParamNo 						:= iSI;
				END_IF  
			END_CASE
    
			ixPNU 			:= ixPNU + 1;   				// count up to next PNU
			
			IF ixPNU < 3 THEN								// if all PNUs are read, goto step 20 and count up the subindex
				IF FML_REF.DeviceType = SFC_DC OR FML_REF.DeviceType = MTR_DCI THEN													(* SFC-DC or MTR-DCI *)
					Step	:= 18;
				ELSE																												(* CMMP-AS or CMMS-AS or CMMS-ST or EMCA-EC or CMMO-ST *)
					Step	:= 20;	
				END_IF
			ELSE            
				Step		:= 22;
			END_IF

		ELSIF FML_REF.Done AND FML_REF.Err THEN
			Status.Err:=TRUE; Status.Cat:=FML_parameter_transfer; Status.ID:=FML_REF.ActValue;
			Step			:= 30;
		END_IF;

	22: // prepare next Subindex 		
		IF (FML_REF.DeviceType = CMMP_AS) 
		OR (FML_REF.DeviceType = CMMS_AS) 
		OR (FML_REF.DeviceType = CMMS_ST) 
		OR (FML_REF.DeviceType = CMMD_AS) 
		OR (FML_REF.DeviceType = SFC_DC) 
		OR (FML_REF.DeviceType = MTR_DCI) THEN		(* CMMP-AS or CMMS_AS or CMMS_ST or CMMD_AS *)	
			IF (DiagBuff[iSI].DiagMsgNumber =  0) 
			OR (ParamNo	= max_iSI)	THEN
				ValidEntries	:= ParamNo;			// if the actual message number is zero or all entries are read, goto step 30
				Status.Err:=FALSE; Status.Cat:=FML_no_category; Status.ID:=FML_no_error;
				Step			:= 30;
			ELSE
				ixPNU	:= 0;					
				Step	:= 20;
			END_IF
		ELSE										(*******EMCA-EC or CMMO-ST*******)
			IF iSI >= max_iSI THEN
				Status.Err:=FALSE; Status.Cat:=FML_no_category; Status.ID:=FML_no_error;
				Step	:= 30;						// if the all entries are read, goto step 30
			ELSE
				ixPNU	:= 0;						// else read the next diagnosis entry (next subindex)
				
				Step	:= 20;
			END_IF
		END_IF
		
		iSI				:= iSI + 1;					// count up the subindex
		
		
	30: (* fill up the rest of the array with FFFF and set Done = TRUE *)
		TimeStart		:= FALSE;
		
		IF ParamNo = 0 THEN
			iSI			:= 1;
		END_IF
		
		FOR iSI := iSI TO maxDiagBuffElements DO
			DiagBuff[iSI].DiagEvent				:= 0;
			DiagBuff[iSI].DiagMsgNumber			:= 16#FFFF;
			DiagBuff[iSI].DiagMsgDescription	:= '';
			DiagBuff[iSI].DiagTimeStamp			:= 0;
			astVisu[iSI].sEvent					:= '';
			astVisu[iSI].sFault 				:= '';
			astVisu[iSI].sStamp 				:= '';
			astVisu[iSI].sText					:= '';
		END_FOR	
   		
		Done			:= TRUE;  							// FB is finished
		Step  			:= 100;
	
	100:(* wait execute to be false *)
		;
END_CASE;


Status.Msg				:= GetStatusMessage(Status);
Error					:= Status.Err;

(* ===== end of function block ============================= *)

END_FUNCTION_BLOCK

// Internal/Blocks/FML_DiagEventString
(* ===============================================================================
   FESTO AG & Co. KG, Esslingen - Copyright 2015. All rights reserved.                       
 ---------------------------------------------------------------------------------
 Functionblock:  FML_DiagEventString 
 Description:    function to get the diagnosis discription of the controller 
 Version:        V 1.0        
 Composer:       Rudolf Schenke 
 Last Update:    10.04.2014                                                                          
------------------------------------------------------------------------------- *)
{library private}
(* ----------------------------------------------------------------------------
Date        Name            	Activity                                                                              
17.03.2013  Rudolf Schenke      created
10.04.2014	Benjamin Kilgus		function name change
10.04.2014	Benjamin Kilgus		events added
=============================================================================== *)
{library public}

FUNCTION FML_DiagEventString : STRING
VAR_INPUT
  dwVal 	: DWORD;		
END_VAR

(*-----------------------------------------------------------
     logic
------------------------------------------------------------*)

CASE dwVal OF 
0:	FML_DiagEventString := 'none';
1:	FML_DiagEventString := 'error';
2:	FML_DiagEventString := 'error gone';
3:	FML_DiagEventString := 'error quit';
4:	FML_DiagEventString := 'overflow timestamp';
5:	FML_DiagEventString := 'warning';
6:	FML_DiagEventString := 'warning gone';
7:	FML_DiagEventString := 'start up event';
8:	FML_DiagEventString := 'configuration';
9:	FML_DiagEventString := 'information';
ELSE;	
	FML_DiagEventString := 'none';
END_CASE

(* ===== end of function ================================== *)

END_FUNCTION

// Internal/Blocks/FaultString/FaultString
(* ===============================================================================
   FESTO AG & Co. KG, Esslingen - Copyright 2015. All rights reserved.                       
 ---------------------------------------------------------------------------------
 Functionblock:  FaultString  
 Description:    function get the error description of the different controllers
 Version:        V 3.5.7.21        
 Composer:       chmm 
 Last Update:    13.11.2017                                                                           
------------------------------------------------------------------------------- *)
{library private}
(* ----------------------------------------------------------------------------
Date        Name            	Activity                                                                              
22.06.2015	Christian Hammer	created
13.11.2017	Christian Hammer	added SFC-DC and MTR-DCI controller
=============================================================================== *)
{library public}

FUNCTION FaultString	:STRING

VAR_INPUT
	iErr 		: DINT;			// error number of the controller
	DeviceType	: INT;			// type of the controller
END_VAR

(* ----- LOGIC -------------------------------------------- *)

CASE DeviceType OF

	(*FaultString for CMMO-ST and EMCA-EC*)
	CMMO_ST,EMCA_EC:
			FaultString	:= ErrorList_CMMO_ST_EMCA_EC(iErr);
	
	(*FaultString for CMMP-AS*)
	CMMP_AS:
			FaultString	:= ErrorList_CMMP_AS(iErr);
			
	(*FaultString for CMMS-AS, CMMS-ST, CMMD-AS *)
	CMMS_AS, CMMS_ST, CMMD_AS:
			FaultString	:= ErrorList_CMMD_CMMS(iErr);

	(*FaultString for SFC_DC, MTR_DCI *)		
	SFC_DC, MTR_DCI:
			FaultString	:= ErrorList_SFC_MTR(iErr);
			
END_CASE

(* ===== end of function ================================== *)

END_FUNCTION

// Internal/Blocks/FaultString/ErrorList_CMMO_ST_EMCA_EC
(* ============================================================================
   FESTO AG & Co. KG, Esslingen - Copyright (c) 2015. All rights reserved.                                   								
  -----------------------------------------------------------------------------  
 Description:    function to get the fault description of the controller CMMO-ST and EMCA-EC 
 Version:		 V3.5.7.21
 Composer:		 chmm
 Last Update:    13.11.2017                                                                           
 ------------------------------------------------------------------------------
Date        Name                Activity                                                                              
22.06.2015	Christian Hammer	created
13.11.2017	Christian Hammer	list updated
============================================================================ *)

FUNCTION ErrorList_CMMO_ST_EMCA_EC : STRING

VAR_INPUT
	iErr	:DINT;			// error number of the controller
END_VAR

(* ----- ASSIGNMENT OF ERROR STRING --------------------------------------- *)

CASE iErr OF
  16#00: ErrorList_CMMO_ST_EMCA_EC := '--';	
  16#01: ErrorList_CMMO_ST_EMCA_EC :='Software error';
  16#02: ErrorList_CMMO_ST_EMCA_EC :='Default parameter file invalid';
  16#03: ErrorList_CMMO_ST_EMCA_EC :='Internal communication error CPUs';
  16#04: ErrorList_CMMO_ST_EMCA_EC :='Non-permitted hardware';
  16#05: ErrorList_CMMO_ST_EMCA_EC :='Zero angle determination';
  16#06: ErrorList_CMMO_ST_EMCA_EC :='Encoder';
  16#07: ErrorList_CMMO_ST_EMCA_EC :='Limit switch positive';
  16#08: ErrorList_CMMO_ST_EMCA_EC :='Limit switch negative';
  16#09: ErrorList_CMMO_ST_EMCA_EC :='Offset determination for current measurement';
  16#0A: ErrorList_CMMO_ST_EMCA_EC :='General error';
  16#0B: ErrorList_CMMO_ST_EMCA_EC :='Parameter file invalid';
  16#0C: ErrorList_CMMO_ST_EMCA_EC :='Firmware update execution error';
  16#0D: ErrorList_CMMO_ST_EMCA_EC :='Overcurrent';
  16#0E: ErrorList_CMMO_ST_EMCA_EC :='I²t malfunction motor';
  16#0F: ErrorList_CMMO_ST_EMCA_EC :='hardware error interface';
  16#10: ErrorList_CMMO_ST_EMCA_EC :='Both limit switches active';
  16#11: ErrorList_CMMO_ST_EMCA_EC :='Softwarelimit positive';
  16#12: ErrorList_CMMO_ST_EMCA_EC :='Softwarelimit negative';
  16#13: ErrorList_CMMO_ST_EMCA_EC :='Positive direction locked';
  16#14: ErrorList_CMMO_ST_EMCA_EC :='Negative direction locked';
  16#15: ErrorList_CMMO_ST_EMCA_EC :='Output stage temperature exceeded';
  16#16: ErrorList_CMMO_ST_EMCA_EC :='Output stage temperature too low';
  16#17: ErrorList_CMMO_ST_EMCA_EC :='Logic voltage exceeded';
  16#18: ErrorList_CMMO_ST_EMCA_EC :='Logic voltage too low';
  16#19: ErrorList_CMMO_ST_EMCA_EC :='Real time error LM-CPU';
  16#1A: ErrorList_CMMO_ST_EMCA_EC :='Intermediate circuit voltage exceeded';
  16#1B: ErrorList_CMMO_ST_EMCA_EC :='Intermediate circuit voltage too low';
  16#1C: ErrorList_CMMO_ST_EMCA_EC :='CAN Node Guarding, FB has master control';
  16#1D: ErrorList_CMMO_ST_EMCA_EC :='CAN bus comm. stopped by master, FB has master control';
  16#1E: ErrorList_CMMO_ST_EMCA_EC :='NetX configuration error';
  16#1F: ErrorList_CMMO_ST_EMCA_EC :='NetX network error';
  16#20: ErrorList_CMMO_ST_EMCA_EC :='FHPP+ incorrect parameterisation';
  16#21: ErrorList_CMMO_ST_EMCA_EC :='FHPP+ incorrect value';
  16#22: ErrorList_CMMO_ST_EMCA_EC :='Homing';
  16#23: ErrorList_CMMO_ST_EMCA_EC :='No index pulse found';
  16#24: ErrorList_CMMO_ST_EMCA_EC :='Drive function is not supported in open-loop operation';
  16#25: ErrorList_CMMO_ST_EMCA_EC :='Path calculation';
  16#26: ErrorList_CMMO_ST_EMCA_EC :='CAN fieldbus parameters missing';
  16#27: ErrorList_CMMO_ST_EMCA_EC :='Save parameters';
  16#28: ErrorList_CMMO_ST_EMCA_EC :='Homing required';
  16#29: ErrorList_CMMO_ST_EMCA_EC :='Target position behind negative software end position';
  16#2A: ErrorList_CMMO_ST_EMCA_EC :='Target position behind positive software end position';
  16#2B: ErrorList_CMMO_ST_EMCA_EC :='Firmware update, invalid firmware';
  16#2C: ErrorList_CMMO_ST_EMCA_EC :='FHPP incorrect record number';
  16#2D: ErrorList_CMMO_ST_EMCA_EC :='I²t warning motor';
  16#2E: ErrorList_CMMO_ST_EMCA_EC :='Index pulse too close on proximity sensor';
  16#2F: ErrorList_CMMO_ST_EMCA_EC :='Following error';
  16#30: ErrorList_CMMO_ST_EMCA_EC :='Braking resistor';
  16#31: ErrorList_CMMO_ST_EMCA_EC :='CVE connection';
  16#32: ErrorList_CMMO_ST_EMCA_EC :='FCT connection with master control';
  16#33: ErrorList_CMMO_ST_EMCA_EC :='Output stage temperature warning';
  16#34: ErrorList_CMMO_ST_EMCA_EC :='Safe Torque Off (STO)';
  16#35: ErrorList_CMMO_ST_EMCA_EC :='CAN Node Guarding, FB does not have master control';
  16#36: ErrorList_CMMO_ST_EMCA_EC :='CAN bus comm. stopped by master, FB does not have master control';
  16#37: ErrorList_CMMO_ST_EMCA_EC :='Standstill monitoring';
  16#38: ErrorList_CMMO_ST_EMCA_EC :='Parameter file access';
  16#39: ErrorList_CMMO_ST_EMCA_EC :='Trace warning';
  16#3A: ErrorList_CMMO_ST_EMCA_EC :='Homing Timeout';
  16#3B: ErrorList_CMMO_ST_EMCA_EC :='Homing method invalid';
  16#3C: ErrorList_CMMO_ST_EMCA_EC :='Two edges in one cycle';
  16#3D: ErrorList_CMMO_ST_EMCA_EC :='Start-up event';
  16#3E: ErrorList_CMMO_ST_EMCA_EC :='Diagnostic memory';
  16#3F: ErrorList_CMMO_ST_EMCA_EC :='Record invalid';
  16#40: ErrorList_CMMO_ST_EMCA_EC :='Last Teaching not successful';
  16#41: ErrorList_CMMO_ST_EMCA_EC :='System reset';
  16#42: ErrorList_CMMO_ST_EMCA_EC :='Address Conflict Detection (ACD)';
  16#43: ErrorList_CMMO_ST_EMCA_EC :='FCT connection without master control';
  16#44: ErrorList_CMMO_ST_EMCA_EC :='Parameter file not compatible with firmware';
  16#45: ErrorList_CMMO_ST_EMCA_EC :='IO-Link system error';
  16#46: ErrorList_CMMO_ST_EMCA_EC :='IO-Link communication error';
  16#47: ErrorList_CMMO_ST_EMCA_EC :='Modbus connection with master control';
  16#48: ErrorList_CMMO_ST_EMCA_EC :='Modbus connection without master control';
  16#49: ErrorList_CMMO_ST_EMCA_EC :='CAN message overflow';
  16#4A: ErrorList_CMMO_ST_EMCA_EC :='Safe Torque Off (STO) discrepancy time';
  16#4B: ErrorList_CMMO_ST_EMCA_EC :='Interpolated Positioning Mode stopped while error occurred on control unit';
  16#4D: ErrorList_CMMO_ST_EMCA_EC :='Value is out of range';
  16#4E: ErrorList_CMMO_ST_EMCA_EC :='Overload 24V outputs';
  16#4F: ErrorList_CMMO_ST_EMCA_EC :='System information';
  16#50: ErrorList_CMMO_ST_EMCA_EC :='EtherCAT connection with master control';
  16#51: ErrorList_CMMO_ST_EMCA_EC :='EtherCAT connection without master control';
  16#52: ErrorList_CMMO_ST_EMCA_EC :='PROFINET connection with master control';
  16#53: ErrorList_CMMO_ST_EMCA_EC :='PROFINET connection without master control';
  16#FF: ErrorList_CMMO_ST_EMCA_EC :='no error';
ELSE
		 ErrorList_CMMO_ST_EMCA_EC := 'Unknown number';
END_CASE;

(* ===== end of function =================================== *)

END_FUNCTION

// Internal/Blocks/FaultString/ErrorList_CMMP_AS
(* ============================================================================
   FESTO AG & Co. KG, Esslingen - Copyright (c) 2015. All rights reserved.                                   								
  -----------------------------------------------------------------------------  
 Description:    function to get the fault description of the controller CMMP-AS 
 Version:		 V1.0
 Composer:		 chmm
 Last Update:    22.06.2015                                                                           
 ------------------------------------------------------------------------------
Date        Name                Activity                                                                              
22.06.2015	Christian Hammer	created
29.02.2016	Christian Hammer	changed String for ID 0 from '' into '--'
============================================================================ *)

FUNCTION ErrorList_CMMP_AS : STRING

VAR_INPUT
	iErr	:DINT;			// error number of the controller
END_VAR

(* ----- ASSIGNMENT OF ERROR STRING --------------------------------------- *)

CASE iErr OF    
  000:       ErrorList_CMMP_AS := '--';
  001:       ErrorList_CMMP_AS := 'Invalid error detected and corrected';
  002:       ErrorList_CMMP_AS := 'Error cleared';
  004:       ErrorList_CMMP_AS := 'Serial number / device type changed (change of modules)';
  007:		 ErrorList_CMMP_AS := 'Consecutive entry';
  008:       ErrorList_CMMP_AS := 'Controller switched on';
  009:       ErrorList_CMMP_AS := 'Controller safety parameters changed';
  010:       ErrorList_CMMP_AS := 'Stack overflow';
  020:       ErrorList_CMMP_AS := 'Intermediate circuit undervoltage';
  030:       ErrorList_CMMP_AS := 'Analogue motor overtemperature';
  031:       ErrorList_CMMP_AS := 'Digital motor overtemperature';
  032:       ErrorList_CMMP_AS := 'Analogue motor overtemperature: broken wire';
  033:       ErrorList_CMMP_AS := 'Analogue motor overtemperature: short circuit';
  040:       ErrorList_CMMP_AS := 'Power section overtemperature';
  041:       ErrorList_CMMP_AS := 'Intermediate circuit overtemperature';
  050:       ErrorList_CMMP_AS := 'Failure of internal voltage 1';
  051:       ErrorList_CMMP_AS := 'Failure of internal voltage 2';
  052:       ErrorList_CMMP_AS := 'Failure of driver supply';
  053:       ErrorList_CMMP_AS := 'Undervoltage of digital I/O';
  054:       ErrorList_CMMP_AS := 'Overcurrent of digital I/O';
  055:       ErrorList_CMMP_AS := 'Module supply voltage failure';
  056:       ErrorList_CMMP_AS := 'X10, [X11] and RS232 supply voltage failure';
  057:       ErrorList_CMMP_AS := 'Safety module internal voltage failure';
  058:       ErrorList_CMMP_AS := 'Failure of Internal voltage 3 (15V)';
  059:       ErrorList_CMMP_AS := 'Encoder supply defective';
  060:       ErrorList_CMMP_AS := 'Output stage short-circuit';
  061:       ErrorList_CMMP_AS := 'Brake chopper overcurrent';
  070:       ErrorList_CMMP_AS := 'Intermediate circuit overvoltage';
  080:       ErrorList_CMMP_AS := 'Resolver angular encoder error';
  081:       ErrorList_CMMP_AS := 'Direction of rotat. of serial and incre. position evaluation is not identical';
  082:       ErrorList_CMMP_AS := 'Incremental encoder Z0 track signals error';
  083:       ErrorList_CMMP_AS := 'Incremental encoder Z1 track signals error';
  084:       ErrorList_CMMP_AS := 'Digital incremental encoder track signals error [X2B]';
  085:       ErrorList_CMMP_AS := 'Incremental encoder Hall generator signals error';
  086:       ErrorList_CMMP_AS := 'Faulty angle encoder communication';
  087:       ErrorList_CMMP_AS := 'Signal amplitude of encoder erroneous [X10]';
  088:       ErrorList_CMMP_AS := 'Internal angle encoder error';
  089:       ErrorList_CMMP_AS := 'Angle encoder at [X2B] not supported';
  090:  	 ErrorList_CMMP_AS := 'Old encoder parameter set';
  091:       ErrorList_CMMP_AS := 'Encoder parameter set cannot be decoded';
  092:       ErrorList_CMMP_AS := 'Unknown encoder parameter set version';
  093:       ErrorList_CMMP_AS := 'Defective data structure angle encoder parameter set';
  094:       ErrorList_CMMP_AS := 'EEPROM data: user-specific configuration faulty';
  095:       ErrorList_CMMP_AS := 'Read/Write error EEPROM parameter data';
  097:       ErrorList_CMMP_AS := 'Encoder EEPROM is write protected';
  098:       ErrorList_CMMP_AS := 'Error in the parameter memory of the angle encoder';
  099:       ErrorList_CMMP_AS := 'Memory size of encoder EEPROM too small';
  100:       ErrorList_CMMP_AS := 'Overspeed';
  110:       ErrorList_CMMP_AS := 'Error when homing is started';
  111:       ErrorList_CMMP_AS := 'Error during homing';
  112:       ErrorList_CMMP_AS := 'Homing: No valid zero pulse';
  113:       ErrorList_CMMP_AS := 'Homing: Timeout';
  114:       ErrorList_CMMP_AS := 'Homing: Incorrect limit switch';
  115:       ErrorList_CMMP_AS := 'Homing: I²t / following error';
  116:       ErrorList_CMMP_AS := 'Homing: End of search path';
  117:       ErrorList_CMMP_AS := 'Homing: Error encoder difference monitoring';
  120:       ErrorList_CMMP_AS := 'CAN: Double node number';
  121:       ErrorList_CMMP_AS := 'CAN: Communication error, bus OFF';
  122:       ErrorList_CMMP_AS := 'CAN: Communication error during transmission';
  123:       ErrorList_CMMP_AS := 'CAN: Communication error during reception';
  124:       ErrorList_CMMP_AS := 'No Node Guarding-telegram received';
  125:       ErrorList_CMMP_AS := 'CAN: RPDO too short';
  129:       ErrorList_CMMP_AS := 'CAN: Protocol error';
  130:       ErrorList_CMMP_AS := 'CAN: Timeout';
  140:       ErrorList_CMMP_AS := 'Autom. current contr. identification: Insufficient intermediate circuit voltage';
  141:       ErrorList_CMMP_AS := 'Autom. current contr. identification: Measurement cycle insufficient';
  142:       ErrorList_CMMP_AS := 'Autom. current contr. identification: Power stage could not be enabled';
  143:       ErrorList_CMMP_AS := 'Autom. current contr. identification: Output stage was switched off prematurely';
  144:       ErrorList_CMMP_AS := 'Autom. angle encoder identification: Encoder type unsuitable';
  145:       ErrorList_CMMP_AS := 'Autom. angle encoder identification: Zero pulse could not be found';
  146:       ErrorList_CMMP_AS := 'Autom. angle encoder identification: Faulty Hall signals';
  147:       ErrorList_CMMP_AS := 'Autom. angle encoder identification: Identification not possible';
  148:       ErrorList_CMMP_AS := 'Autom. angle encoder identification: Invalid number of pairs of poles';
  149:       ErrorList_CMMP_AS := 'Autom. parameter identification: General error';
  150:       ErrorList_CMMP_AS := 'Division by zero';
  151:       ErrorList_CMMP_AS := 'Mathematical overflow during division';
  152:       ErrorList_CMMP_AS := 'Mathematical underflow';
  160:       ErrorList_CMMP_AS := 'Error during program execution';
  161:       ErrorList_CMMP_AS := 'Illegal interrupt';
  162:       ErrorList_CMMP_AS := 'Initialisation error';
  163:       ErrorList_CMMP_AS := 'Unexpected state';
  170:       ErrorList_CMMP_AS := 'Following error limit exceeded';
  171:       ErrorList_CMMP_AS := 'Encoder difference monitoring';
  172:       ErrorList_CMMP_AS := 'Current jump control';
  173:       ErrorList_CMMP_AS := 'Speed jump safety module monitoring';
  180:       ErrorList_CMMP_AS := 'Analogue motor temperature';
  181:       ErrorList_CMMP_AS := 'Temperature power stage';
  190:       ErrorList_CMMP_AS := 'reserved (CMMS)';
  200:       ErrorList_CMMP_AS := 'External error request via DIN';
  210:       ErrorList_CMMP_AS := 'Error 1 current measurement U';
  211:       ErrorList_CMMP_AS := 'Error 1 current measurement V';
  212:       ErrorList_CMMP_AS := 'Error 2 current measurement U';
  213:       ErrorList_CMMP_AS := 'Error 2 current measurement V';
  220:       ErrorList_CMMP_AS := 'PROFIBUS: Initialisation error';
  221:       ErrorList_CMMP_AS := 'PROFIBUS: reserved';
  222:       ErrorList_CMMP_AS := 'PROFIBUS: Faulty communication';
  223:       ErrorList_CMMP_AS := 'PROFIBUS: Invalid slave address';
  224:       ErrorList_CMMP_AS := 'PROFIBUS: Conversion error';
  225:       ErrorList_CMMP_AS := 'PROFIBUS: Access violation';
  230:       ErrorList_CMMP_AS := 'Actual position: No valid record available';
  231:       ErrorList_CMMP_AS := 'Actual position: Invalid checksum';
  232:       ErrorList_CMMP_AS := 'Actual position: Flash content inconsistent';
  250:       ErrorList_CMMP_AS := 'Invalid device type';
  251:       ErrorList_CMMP_AS := 'Device type not supported';
  252:       ErrorList_CMMP_AS := 'Invalid hardware revision';
  253:       ErrorList_CMMP_AS := 'Device with restricted functionality: Firmware cannot be executed';
  254:       ErrorList_CMMP_AS := 'Invalid power stage type';
  255:       ErrorList_CMMP_AS := 'Incompatibility FW/HW';
  260:       ErrorList_CMMP_AS := 'Missing user parameter set';
  261:       ErrorList_CMMP_AS := 'Checksum error';
  262:       ErrorList_CMMP_AS := 'Flash: Error when writing';
  263:       ErrorList_CMMP_AS := 'Flash: Error during deletion';
  264:       ErrorList_CMMP_AS := 'Flash: Internal flash error';
  265:       ErrorList_CMMP_AS := 'Missing calibration data';
  266:       ErrorList_CMMP_AS := 'Missing position data sets';
  267:       ErrorList_CMMP_AS := 'Faulty data tables (CAM)';
  270:       ErrorList_CMMP_AS := 'Following error warning threshold';
  280:       ErrorList_CMMP_AS := 'Missing operating hour meter';
  281:       ErrorList_CMMP_AS := 'Operating hour counter: Write error';
  282:       ErrorList_CMMP_AS := 'Operating hour counter corrected';
  283:       ErrorList_CMMP_AS := 'Operating hour counter converted';
  290:       ErrorList_CMMP_AS := 'Memory card not available';
  291:       ErrorList_CMMP_AS := 'Memory card: Initialisation error';
  292:       ErrorList_CMMP_AS := 'Memory card: Data error';
  293:       ErrorList_CMMP_AS := 'Memory card: Write error';
  294:       ErrorList_CMMP_AS := 'Memory card: Firmware download error';
  300:       ErrorList_CMMP_AS := 'Internal conversion error';
  310:       ErrorList_CMMP_AS := 'Motor I²t';
  311:       ErrorList_CMMP_AS := 'Power stage I²t';
  312:       ErrorList_CMMP_AS := 'PFC I²t';
  313:       ErrorList_CMMP_AS := 'Braking resistor I²t';
  314:       ErrorList_CMMP_AS := 'I²t active power overload';
  320:       ErrorList_CMMP_AS := 'Intermediate circuit charging time exceeded';
  321:       ErrorList_CMMP_AS := 'Undervoltage for active PFC';
  325:       ErrorList_CMMP_AS := 'Brake chopper overload';
  326:       ErrorList_CMMP_AS := 'Intermediate circuit discharge time exceeded';
  327:       ErrorList_CMMP_AS := 'Power supply missing for controller enable';
  328:       ErrorList_CMMP_AS := 'Power supply failure during controller enable';
  329:       ErrorList_CMMP_AS := 'Phase failure';
  330:       ErrorList_CMMP_AS := 'Encoder emulation following error';
  340:       ErrorList_CMMP_AS := 'No synchronisation via field bus';
  341:       ErrorList_CMMP_AS := 'Field bus synchronisation error';
  350:       ErrorList_CMMP_AS := 'Linear motor spinning protection';
  351:       ErrorList_CMMP_AS := 'reserved (CMMS)';
  355:       ErrorList_CMMP_AS := 'Error during the determination of the commutation position';
  360:       ErrorList_CMMP_AS := 'Parameter was limited';
  361:       ErrorList_CMMP_AS := 'Parameter was not accepted';
  370:  	 ErrorList_CMMP_AS := 'SERCOS: Excessive distortion';
  371:       ErrorList_CMMP_AS := 'SERCOS: Ring not closed';
  372:       ErrorList_CMMP_AS := 'SERCOS: MST missing twice';
  373:       ErrorList_CMMP_AS := 'SERCOS: Illegal phase requested by master';
  374:       ErrorList_CMMP_AS := 'SERCOS: MDT missing twice';
  375:       ErrorList_CMMP_AS := 'SERCOS: Unknown operation mode selected';
  376:       ErrorList_CMMP_AS := 'SERCOS: T3 invalid';
  377:       ErrorList_CMMP_AS := 'SERCOS field bus';
  380:  	 ErrorList_CMMP_AS := 'SERCOS: SERCON Status event';
  381:  	 ErrorList_CMMP_AS := 'SERCOS: No module';
  382:  	 ErrorList_CMMP_AS := 'SERCOS: Defective module';
  383:  	 ErrorList_CMMP_AS := 'SERCOS: S-0-0127: Invalid data in S-0-0021';
  384:  	 ErrorList_CMMP_AS := 'SERCOS: S-0-0127: Illegal IDNs in AT or MDT';
  385:  	 ErrorList_CMMP_AS := 'SERCOS: S-0-0128: Invalid data in S-0-0022';
  386:  	 ErrorList_CMMP_AS := 'SERCOS: S-0-0128: Invalid scaling';
  387:  	 ErrorList_CMMP_AS := 'SERCOS: Invalid IDN in S-0-0026 / S-0-0027';
  388:  	 ErrorList_CMMP_AS := 'SERCOS: Error at conversion';
  389:  	 ErrorList_CMMP_AS := 'SERCOS: SERCON 410b mode activated';
  390:  	 ErrorList_CMMP_AS := 'SERCOS: List S-0-0370: Invalid configuration MDT-Data container';
  391:  	 ErrorList_CMMP_AS := 'SERCOS: List S-0-0371: Invalid configuration AT-Data container';
  392:  	 ErrorList_CMMP_AS := 'SERCOS: Cyclic channel fault MDT';
  393:  	 ErrorList_CMMP_AS := 'SERCOS: Cyclic channel fault AT';
  394:  	 ErrorList_CMMP_AS := 'SERCOS: Cyclic data container fault MDT';
  395:  	 ErrorList_CMMP_AS := 'SERCOS: Cyclic data container fault AT';
  400:       ErrorList_CMMP_AS := 'Negative software limit reached';
  401:       ErrorList_CMMP_AS := 'Positive software limit reached';
  402:       ErrorList_CMMP_AS := 'Positioning beyond negative software limit switch suppressed';
  403:       ErrorList_CMMP_AS := 'Positioning beyond positive software limit switch suppressed';
  410:  	 ErrorList_CMMP_AS := 'Record sequence: Synchronisation error';
  418:  	 ErrorList_CMMP_AS := 'reserved (CMMS)';
  419:  	 ErrorList_CMMP_AS := 'reserved (CMMS)';
  420:       ErrorList_CMMP_AS := 'Positioning: Drive stops automatically because there is no follow-up positioning';
  421:       ErrorList_CMMP_AS := 'Positioning: Drive stops as rotation reversal is not allowed';
  422:       ErrorList_CMMP_AS := 'Positioning: Illegal rotation reversal after "stop"';
  423:       ErrorList_CMMP_AS := 'Start positioning rejected: Wrong mode of operation';
  424:       ErrorList_CMMP_AS := 'Please enforce homing run!';
  425:       ErrorList_CMMP_AS := 'Rotary axis: Direction of rotation is not allowed';
  429:  	 ErrorList_CMMP_AS := 'Error at starting the positioning';
  430:       ErrorList_CMMP_AS := 'Limit switch: Negative setpoint value blocked';
  431:       ErrorList_CMMP_AS := 'Limit switch: Positive setpoint value blocked';
  432:       ErrorList_CMMP_AS := 'Limit switch: Positioning suppressed';
  433:  	 ErrorList_CMMP_AS := 'reserved';
  434:  	 ErrorList_CMMP_AS := 'reserved (CMMS)';
  440:  	 ErrorList_CMMP_AS := 'Error in Cam data tables';
  441:  	 ErrorList_CMMP_AS := 'Cam Disc: General error homing';
  450:       ErrorList_CMMP_AS := 'Driver supply cannot be switched off';
  451:       ErrorList_CMMP_AS := 'Driver supply cannot be activated';
  452:       ErrorList_CMMP_AS := 'Driver supply was activated';
  453:  	 ErrorList_CMMP_AS := 'reserved (CMMS)';
  470:       ErrorList_CMMP_AS := 'Timeout setup mode';
  480:  	 ErrorList_CMMP_AS := 'Please enforce homing run!';
  491:  	 ErrorList_CMMP_AS := 'DCO file: wrong password';
  492:  	 ErrorList_CMMP_AS := 'DCO file: Data error';
  500:  	 ErrorList_CMMP_AS := 'Too many synchronous PDOs';
  501:  	 ErrorList_CMMP_AS := 'SDO error has occurred';
  510:  	 ErrorList_CMMP_AS := 'Unknown Safety module or driver supply defective';
  511:  	 ErrorList_CMMP_AS := 'Safety function: Driver supply defective';
  512:  	 ErrorList_CMMP_AS := 'Safety module: Dissimilar module type';
  513:  	 ErrorList_CMMP_AS := 'Safety module: Dissimilar  module version';
  514:  	 ErrorList_CMMP_AS := 'Safety module: SSIO communication error';
  515:  	 ErrorList_CMMP_AS := 'Safety module: Brake control error';
  516:  	 ErrorList_CMMP_AS := 'Safety module: Dissimilar serial number';
  520:  	 ErrorList_CMMP_AS := 'Safety function: Error';
  521:  	 ErrorList_CMMP_AS := 'Safety function: Discrepancy time expired';
  522:  	 ErrorList_CMMP_AS := 'Safety function: Failure of driver supply with active PWM control';
  523:  	 ErrorList_CMMP_AS := 'Safety module: Overlapping velocity limits in basic unit';
  524..529:	 ErrorList_CMMP_AS := 'Safety function: Error';
  530:  	 ErrorList_CMMP_AS := 'USF0: Safety condition violated';
  531:  	 ErrorList_CMMP_AS := 'USF1: Safety condition violated';
  532:  	 ErrorList_CMMP_AS := 'USF2: Safety condition violated';
  533:  	 ErrorList_CMMP_AS := 'USF3: Safety condition violated';
  534:  	 ErrorList_CMMP_AS := 'not used';
  535:  	 ErrorList_CMMP_AS := 'not used';
  536:  	 ErrorList_CMMP_AS := 'SDI0: Safety condition violated';
  537:  	 ErrorList_CMMP_AS := 'SDI1: Safety condition violated';
  538:  	 ErrorList_CMMP_AS := 'SLI0: Safety condition violated';
  539:  	 ErrorList_CMMP_AS := 'SLI1: Safety condition violated';
  540:  	 ErrorList_CMMP_AS := 'SBC: Safety condition violated';
  541:  	 ErrorList_CMMP_AS := 'SBT: Safety condition violated';
  542:  	 ErrorList_CMMP_AS := 'SS2: Safety condition violated';
  543:  	 ErrorList_CMMP_AS := 'SOS: Safety condition violated';
  544:  	 ErrorList_CMMP_AS := 'SS1: Safety condition violated';
  545:  	 ErrorList_CMMP_AS := 'STO: Safety condition violated';
  546:  	 ErrorList_CMMP_AS := 'SBC: Brake not released for > 24h';
  547:  	 ErrorList_CMMP_AS := 'SOS: SOS requested for > 24 h';
  548:  	 ErrorList_CMMP_AS := 'not used';
  549:  	 ErrorList_CMMP_AS := 'not used';
  550:  	 ErrorList_CMMP_AS := 'No actual speed / position value available or standstill for > 24 h';
  551:  	 ErrorList_CMMP_AS := 'SINCOS encoder [X2B] - signal error';
  552:  	 ErrorList_CMMP_AS := 'SINCOS encoder [X2B] - standstill > 24 h';
  553:  	 ErrorList_CMMP_AS := 'Resolver [X2A] - signal error';
  554:  	 ErrorList_CMMP_AS := 'EnDat encoder [X2B] - sensor error';
  555:  	 ErrorList_CMMP_AS := 'EnDat encoder [X2B] - wrong sensor / type';
  556:  	 ErrorList_CMMP_AS := 'Incremental encoder X10 - signal error';
  557:  	 ErrorList_CMMP_AS := 'Other encoder [X2B] - Faulty angle information';
  558:  	 ErrorList_CMMP_AS := 'Impermissible acceleration detected';
  559..564:	 ErrorList_CMMP_AS := 'not used';
  565:  	 ErrorList_CMMP_AS := 'Angle sensor error (others)';
  566:  	 ErrorList_CMMP_AS := 'Homing error';
  567:  	 ErrorList_CMMP_AS := 'Wrong homing method';
  568:  	 ErrorList_CMMP_AS := 'Speed / angle difference encoder 1 - 2';
  569:  	 ErrorList_CMMP_AS := 'Error Cross comparison encoder evaluation';
  570:  	 ErrorList_CMMP_AS := 'Self test I/O error (internal/external)';
  571:  	 ErrorList_CMMP_AS := 'Digital inputs - wrong signal level';
  572:  	 ErrorList_CMMP_AS := 'Digital inputs - missing test pulse';
  573:  	 ErrorList_CMMP_AS := 'Analogue input error (value range)';
  574:  	 ErrorList_CMMP_AS := 'Error at current measuring';
  575:  	 ErrorList_CMMP_AS := 'Error at motor voltage measuring';
  576:  	 ErrorList_CMMP_AS := 'Electronic temperature too high';
  577:	 	 ErrorList_CMMP_AS := 'not used';
  578:	 	 ErrorList_CMMP_AS := 'not used';
  579:	 	 ErrorList_CMMP_AS := 'not used';
  580:  	 ErrorList_CMMP_AS := 'Plausibility check parameters';
  581:  	 ErrorList_CMMP_AS := 'General error parameterisation';
  582..583:	 ErrorList_CMMP_AS := 'not used';
  584:  	 ErrorList_CMMP_AS := 'Buffer internal communication';
  585:  	 ErrorList_CMMP_AS := 'Communication safety module - base unit';
  586:  	 ErrorList_CMMP_AS := 'Cross comparison error processor 1 - 2';
  587..590:	 ErrorList_CMMP_AS := 'not used';
  591:  	 ErrorList_CMMP_AS := 'Failsafe supply/safe pulse inhibitor';
  592:  	 ErrorList_CMMP_AS := 'External voltage supply error';
  593:  	 ErrorList_CMMP_AS := 'Internal voltage supply error';
  594:  	 ErrorList_CMMP_AS := 'Error management: Too many errors';
  595:  	 ErrorList_CMMP_AS := 'Diagnosis Memory writing error';
  596:  	 ErrorList_CMMP_AS := 'Error on saving parameter set';
  597:  	 ErrorList_CMMP_AS := 'FLASH checksum error';
  598:  	 ErrorList_CMMP_AS := 'Internal monitoring processor 1 - 2';
  599:  	 ErrorList_CMMP_AS := 'Other unexpected error';
  600..610:  ErrorList_CMMP_AS := 'User-specific error ethernet module';
  620:  	 ErrorList_CMMP_AS := 'EtherCAT: Initialisation error';
  621:  	 ErrorList_CMMP_AS := 'EtherCAT: Initialisation error';
  622:  	 ErrorList_CMMP_AS := 'EtherCAT: Protocol error';
  623:  	 ErrorList_CMMP_AS := 'EtherCAT: Invalid RPDO length';
  624:  	 ErrorList_CMMP_AS := 'EtherCAT: Invalid TPDO length';
  625:  	 ErrorList_CMMP_AS := 'EtherCAT: Erroneous cyclic communication';
  630:  	 ErrorList_CMMP_AS := 'EtherCAT: Defective module';
  631:  	 ErrorList_CMMP_AS := 'EtherCAT: Invalid data';
  632:  	 ErrorList_CMMP_AS := 'EtherCAT: TPDO data has not been read';
  633:  	 ErrorList_CMMP_AS := 'EtherCAT: No distributed clocks active';
  634:  	 ErrorList_CMMP_AS := 'EtherCAT: Missing SYNC message in IPO cycle';
  640:  	 ErrorList_CMMP_AS := 'DeviceNet: Duplicate MAC ID';
  641:  	 ErrorList_CMMP_AS := 'DeviceNet: Bus power lost';
  642:  	 ErrorList_CMMP_AS := 'DeviceNet: RX queue overflow';
  643:  	 ErrorList_CMMP_AS := 'DeviceNet: TX queue overflow';
  644:  	 ErrorList_CMMP_AS := 'DeviceNet: IO message not sent';
  645:  	 ErrorList_CMMP_AS := 'DeviceNet: Bus OFF';
  646:  	 ErrorList_CMMP_AS := 'DeviceNet: CAN controller overflow';
  650:  	 ErrorList_CMMP_AS := 'DeviceNet active, but no module';
  651:  	 ErrorList_CMMP_AS := 'Timeout IO connection';
  660:  	 ErrorList_CMMP_AS := 'Modbus/TCP: No free TCP/IP instances';
  670:  	 ErrorList_CMMP_AS := 'Modbus/TCP: Timeout TCP/IP';
  671:  	 ErrorList_CMMP_AS := 'Modbus/TCP: Timeout Modbus TCP/IP';
  672:  	 ErrorList_CMMP_AS := 'Modbus/TCP: Buffer overflow';
  673:  	 ErrorList_CMMP_AS := 'Modbus/TCP: Telegram length too short';
  674:  	 ErrorList_CMMP_AS := 'Modbus/TCP: Telegram length too long';
  680:  	 ErrorList_CMMP_AS := 'EtherNet/IP: Serious fault';
  681:  	 ErrorList_CMMP_AS := 'EtherNet/IP: General communication fault';
  682:  	 ErrorList_CMMP_AS := 'EtherNet/IP: Connection closed';
  683:  	 ErrorList_CMMP_AS := 'EtherNet/IP: Connection aborted';
  684:  	 ErrorList_CMMP_AS := 'EtherNet/IP: Duplicate network address';
  690:  	 ErrorList_CMMP_AS := 'EtherNet/IP: Duplicate network address';
  691:  	 ErrorList_CMMP_AS := 'EtherNet/IP: Incorrect IP configuration';
  692:  	 ErrorList_CMMP_AS := 'EtherNet/IP: Field bus module not found';
  693:  	 ErrorList_CMMP_AS := 'EtherNet/IP: Module version not supported';
  701:  	 ErrorList_CMMP_AS := 'FHPP: Mathematical error';
  702:  	 ErrorList_CMMP_AS := 'FHPP: Factor group invalid';
  703:  	 ErrorList_CMMP_AS := 'FHPP: Invalid operating mode change';
  711:  	 ErrorList_CMMP_AS := 'FHPP: Wrong receive telegram length';
  712:  	 ErrorList_CMMP_AS := 'FHPP: Wrong response telegram length';
  720:  	 ErrorList_CMMP_AS := 'PROFINET: Initialising error';
  721:  	 ErrorList_CMMP_AS := 'PROFINET: Bus error';
  723:  	 ErrorList_CMMP_AS := 'PROFINET: Invalid IP configuration';
  724:  	 ErrorList_CMMP_AS := 'PROFINET: Invalid Device name';
  725:  	 ErrorList_CMMP_AS := 'PROFINET: Module faulty';
  726:  	 ErrorList_CMMP_AS := 'PROFINET: Indication invalid/not supported';
  730:  	 ErrorList_CMMP_AS := 'PROFIenergy: State not possible';
  780:  	 ErrorList_CMMP_AS := 'NRT frame can not be send';
  800:       ErrorList_CMMP_AS := 'Overflow current controller IRQ';
  801:       ErrorList_CMMP_AS := 'Overflow speed controller IRQ';
  802:       ErrorList_CMMP_AS := 'Overflow position controller IRQ';
  803:       ErrorList_CMMP_AS := 'Overflow interpolator IRQ';
  814:       ErrorList_CMMP_AS := 'Overflow low-level IRQ';
  815:       ErrorList_CMMP_AS := 'Overflow MDC IRQ';
  820:       ErrorList_CMMP_AS := 'Internal sequencing control: Event';
  821:  	 ErrorList_CMMP_AS := 'Multiple-started KO write access';
  830:       ErrorList_CMMP_AS := 'Invalid module';
  831:       ErrorList_CMMP_AS := 'Module not supported';
  832:       ErrorList_CMMP_AS := 'Module: Hardware revision not supported';
  833:       ErrorList_CMMP_AS := 'Module: Write error';
  834:  	 ErrorList_CMMP_AS := 'MC2000 Watchdog';
  840:  	 ErrorList_CMMP_AS := 'Conditions for controller enable not fulfilled';
  900:       ErrorList_CMMP_AS := 'External RAM not recognized';
  901:       ErrorList_CMMP_AS := 'External flash not recognized';
  902:       ErrorList_CMMP_AS := 'Error at FPGA boot-up';
  903:       ErrorList_CMMP_AS := 'Error at SD-ADU start';
  904:       ErrorList_CMMP_AS := 'SD-ADU synchronisation error after start';
  905:       ErrorList_CMMP_AS := 'SD-ADU not synchronous';
  906:       ErrorList_CMMP_AS := 'IRQ0 (current controller): Trigger error';
  907:  	 ErrorList_CMMP_AS := 'Missing CAN controller';
  908:  	 ErrorList_CMMP_AS := 'Checksum error in device parameters';
  909:       ErrorList_CMMP_AS := 'Illegal firmware version';
  910:       ErrorList_CMMP_AS := 'Internal insitialising error';
  911:  	 ErrorList_CMMP_AS := 'Memory error when copying';
  912:  	 ErrorList_CMMP_AS := 'Error when reading the controller/power section coding';
  913:  	 ErrorList_CMMP_AS := 'Software initialisation error';
  920:  	 ErrorList_CMMP_AS := 'Error during firmware download';
  921:  	 ErrorList_CMMP_AS := 'Error during bootloader update';
ELSE
     		 ErrorList_CMMP_AS := 'no text for the specified number';
END_CASE;

END_FUNCTION

// Internal/Blocks/FaultString/ErrorList_CMMD_CMMS
(* ============================================================================
   FESTO AG & Co. KG, Esslingen - Copyright (c) 2015. All rights reserved.                                   								
  -----------------------------------------------------------------------------  
 Description:    function to get the fault description of the controller CMMD-AS 
 Version:		 V1.0
 Composer:		 chmm
 Last Update:    22.06.2015                                                                           
 ------------------------------------------------------------------------------
Date        Name                Activity                                                                              
22.06.2015	Christian Hammer	created
29.02.2016	Christian Hammer	changed String for ID 0 from '' into '--'
============================================================================ *)

FUNCTION ErrorList_CMMD_CMMS : STRING

VAR_INPUT
	iErr	:DINT;			// error number of the controller
END_VAR

(* ----- ASSIGNMENT OF ERROR STRING --------------------------------------- *)

CASE iErr OF
	  16#0:   	ErrorList_CMMD_CMMS := '--';
	  16#06180: ErrorList_CMMD_CMMS := 'Stack Overflow';
	  16#03220: ErrorList_CMMD_CMMS := 'Undervoltage in intermediate circuit';
	  16#04310: ErrorList_CMMD_CMMS := 'Temperature monitoring, motor';
	  16#04210: ErrorList_CMMD_CMMS := 'Excess/low temperature of power electronics';
	  16#05114: ErrorList_CMMD_CMMS := '5 V electronics supply fault';
	  16#05115: ErrorList_CMMD_CMMS := 'Error in 24 V supply';
	  16#08000: ErrorList_CMMD_CMMS := 'Error in driver supply';
	  16#02320: ErrorList_CMMD_CMMS := 'Over-current of the intermediate circuit/output stage';
	  16#03210: ErrorList_CMMD_CMMS := 'Overvoltage in intermediate circuit';
	  16#07386: ErrorList_CMMD_CMMS := 'Angle encoder communication fault';
	  16#07388: ErrorList_CMMD_CMMS := 'Internal angle encoder error';
	  16#08A81: ErrorList_CMMD_CMMS := 'Homing error';
	  16#08181: ErrorList_CMMD_CMMS := 'CAN: general error';
	  16#08130: ErrorList_CMMD_CMMS := 'CAN: TIME-out Nodeguarding';
	  16#06197: ErrorList_CMMD_CMMS := 'Error, motor identification';
	  16#06187: ErrorList_CMMD_CMMS := 'Initialisation fault';
	  16#06183: ErrorList_CMMD_CMMS := 'Unexpected status / programming error';    
	  16#08611: ErrorList_CMMD_CMMS := 'Following error monitoring';   
	  16#04280: ErrorList_CMMD_CMMS := 'Output stage temperature 5°C below maximum';
	  16#02380: ErrorList_CMMD_CMMS := 'I²t at 80%';
	  16#05210: ErrorList_CMMD_CMMS := 'Error, offset current measurement';
	  16#07500: ErrorList_CMMD_CMMS := 'Error in PROFIBUS initialisation';
	  16#06081: ErrorList_CMMD_CMMS := 'Incorrect firmware';
	  16#05581: ErrorList_CMMD_CMMS := 'Checksum error';
	  16#07680: ErrorList_CMMD_CMMS := 'No SD available';
	  16#07681: ErrorList_CMMD_CMMS := 'SD initialisation error';
	  16#07682: ErrorList_CMMD_CMMS := 'SD parameter set error';
	  16#02312: ErrorList_CMMD_CMMS := 'I²t-error motor (I²t at 100%)';
	  16#02311: ErrorList_CMMD_CMMS := 'I²t-error controller (I²t at 100%)';
	  16#03280: ErrorList_CMMD_CMMS := 'Intermediate circuit charging time exceeded';
	  16#03285: ErrorList_CMMD_CMMS := 'Power supply failure during controller enable';
	  16#06199: ErrorList_CMMD_CMMS := 'Time out with fast stop';
	  16#08612: ErrorList_CMMD_CMMS := 'Limit switch error or software limit error';  
	  16#06193: ErrorList_CMMD_CMMS := 'Path program error, unknown command';
	  16#06192: ErrorList_CMMD_CMMS := 'Error in path program jump destination';
	  16#08681: ErrorList_CMMD_CMMS := 'Positioning: Error in pre-computation';
	  16#08600: ErrorList_CMMD_CMMS := 'Message, homing required';
	  16#06191: ErrorList_CMMD_CMMS := 'Error in position data record';
	  16#08087: ErrorList_CMMD_CMMS := 'DIN4 plausibility error';
	  16#07582: ErrorList_CMMD_CMMS := 'DeviceNet communication';
	  16#07584: ErrorList_CMMD_CMMS := 'DeviceNet general error';
	  16#06195: ErrorList_CMMD_CMMS := 'General arithmetic error';
	  16#06380: ErrorList_CMMD_CMMS := 'Operating mode error';
	  16#07510: ErrorList_CMMD_CMMS := 'RS232 communication error';
ELSE
  				ErrorList_CMMD_CMMS := 'Unknown number';
END_CASE;

(* ===== end of function =================================== *)

END_FUNCTION

// Internal/Blocks/FaultString/ErrorList_SFC_MTR
(* ============================================================================
   FESTO AG & Co. KG, Esslingen - Copyright (c) 2015. All rights reserved.                                   								
  -----------------------------------------------------------------------------  
 Description:    function to get the fault description of the controller SFC-DC and MTR-DCI 
 Version:		 V1.0
 Composer:		 chmm
 Last Update:    21.11.2017                                                                           
 ------------------------------------------------------------------------------
Date        Name                Activity                                                                              
21.11.2017	Christian Hammer	created
============================================================================ *)

FUNCTION ErrorList_SFC_MTR : STRING

VAR_INPUT
	iErr	:DINT;			// error number of the controller
END_VAR

(* ----- ASSIGNMENT OF ERROR STRING --------------------------------------- *)

CASE iErr OF
	000:   	ErrorList_SFC_MTR := '--';
	031:   	ErrorList_SFC_MTR := 'Position error';
	106:   	ErrorList_SFC_MTR := 'Motor stop';
	032:   	ErrorList_SFC_MTR := 'Homing error';
	101:   	ErrorList_SFC_MTR := 'Overheating';
	070:   	ErrorList_SFC_MTR := 'Load power down';
	100:   	ErrorList_SFC_MTR := 'I2t error';
	052:   	ErrorList_SFC_MTR := 'Hardware error';
	002:   	ErrorList_SFC_MTR := 'Target position out of limit';
	003:   	ErrorList_SFC_MTR := 'Illegar record';
	001:   	ErrorList_SFC_MTR := 'Please enforce homing run';
	035:   	ErrorList_SFC_MTR := 'Position plausibility error';
	071:   	ErrorList_SFC_MTR := 'Digital power down';
	103:   	ErrorList_SFC_MTR := 'Motor error';
	036:   	ErrorList_SFC_MTR := 'Standstill';
	051:   	ErrorList_SFC_MTR := 'CAN bus error';

	  
ELSE
  			ErrorList_SFC_MTR := 'Unknown number';
END_CASE;

(* ===== end of function =================================== *)

END_FUNCTION

// Internal/Blocks/FML_TimeStamp
(* ===============================================================================
   FESTO AG & Co. KG, Esslingen - Copyright 2015. All rights reserved.                       
 ---------------------------------------------------------------------------------
 Functionblock:  FML_TimeStamp
 Description:    function to build a typical FML_TimeStamp from raw time value 'nnd:hh:mm:ss:uuu' 
 Version:        V 1.0        
 Composer:       Rudolf Schenke 
 Last Update:    10.04.2014                                                                          
------------------------------------------------------------------------------- *)
{library private}
(* ----------------------------------------------------------------------------
Date        Name            	Activity                                                                              
17.03.2013  Rudolf Schenke      created
10.04.2014	Benjamin Kilgus		function name change
=============================================================================== *)
{library public}


FUNCTION FML_TimeStamp : STRING
VAR_INPUT	
  	dwTime  	: UDINT;	// time
	uiExponent 	: USINT;	// exponent if dwTime differ from unit ms z.B. 0.01, 0.1, 0, 10, 100    
END_VAR
VAR
  	dwTemp 		: DWORD;
END_VAR

(*-----------------------------------------------------------
     logic
------------------------------------------------------------*)

IF uiExponent = 0 THEN
	uiExponent := 1;
END_IF
//dwTime := dwTime * uiExponent;
//dwTemp := dwTime / (1000 * 3600 * 24); 			// days
//FML_TimeStamp := FormatInt(dwTemp, '%i1t:');

dwTime := dwTime MOD (1000 * 3600 * 24);
dwTemp := dwTime / (3600 * 1000);        			// hours
//FML_TimeStamp := CONCAT(FML_TimeStamp, FormatInt(dwTemp, '%i2:'));
FML_TimeStamp := FormatInt(dwTemp, '%i2:');

dwTime := dwTime MOD (3600 * 1000);
dwTemp := dwTime / (60 * 1000);          			// minutes
FML_TimeStamp := CONCAT(FML_TimeStamp, FormatInt(dwTemp, '%i2:'));

dwTime := dwTime MOD (60 * 1000);
dwTemp := dwTime / 1000;          					// seconds
FML_TimeStamp := CONCAT(FML_TimeStamp, FormatInt(dwTemp, '%i2.'));

dwTime := dwTime MOD (1000);
FML_TimeStamp := CONCAT(FML_TimeStamp, FormatInt(dwTime, '%i3'));

(* ===== end of function ================================== *)

END_FUNCTION

// Internal/Blocks/FormatInt
(* ===============================================================================
   FESTO AG & Co. KG, Esslingen - Copyright 2015. All rights reserved.                       
 ---------------------------------------------------------------------------------
 Functionblock:  FML_TimeStamp
 Description:    function to format INT or UINT variables into string
 Version:        V 1.0        
 Composer:       Rudolf Schenke 
 Last Update:    21.05.2013                                                                          
------------------------------------------------------------------------------- *)
{library private}
(* ----------------------------------------------------------------------------
Date        Name            	Activity                                                                              
21.05.2013  Rudolf Schenke      created
=============================================================================== *)
{library public}

FUNCTION FormatInt : STRING
VAR_INPUT
  	value : UDINT;
  	fm    : STRING;  
END_VAR

VAR
  	iWidth  : INT;      	// width of formatted value
  	iPosi   : INT;      	// position of format %mn
 	sType   : STRING;   	 
 	diVal   : DINT; 
 	uiVal   : UDINT;
	Char    : UCHAR;
END_VAR

(* Formatting part = %in for INT  values (with opt. - 
                     %un for UINT values
                     %xn for hex notation
     with n > 0 => length of the formatted value
          n = 0 => length of ..._TO_STRING result
*)

(*-----------------------------------------------------------
     logic
------------------------------------------------------------*)

IF len(fm) < 3 THEN       					// minimum length = 3
  FormatInt := '';
  RETURN;
END_IF
iPosi := Find(fm, '%');   					// position of formatting part
IF iPosi = 0 THEN
  FormatInt := '';
  RETURN;
END_IF

sType := mid(fm,1,iPosi+1);                 // type = i | u | x
iWidth := STRING_TO_INT(MID(fm,1,iPosi+2)); // width

IF sType =  'i' THEN  						// ---- integer - with opt. minus-sign --
  diVal := UDINT_TO_DINT(value);
  sType := DINT_TO_STRING(diVal);
ELSIF sType = 'u' THEN  					// ---- unsigned int -----
  uiVal := value;
  sType := UDINT_TO_STRING(uiVal);
ELSIF sType = 'x' THEN
  sType := '';
  uiVal := value;
  WHILE uiVal <> 0 DO
    Char.char  := UDINT_TO_BYTE((uiVal AND 15) + 48);
    IF Char.char > 57 THEN
      Char.char := Char.char + 7;
		END_IF
    sType := CONCAT(Char.str, sType);
    uiVal := SHR(uiVal,4);
	END_WHILE
END_IF

IF iWidth <> 0 THEN
  WHILE len(sType) < (iWidth) DO
    sType := CONCAT('0', sType);
  END_WHILE
END_IF

FormatInt := REPLACE(fm,sType,3,iPosi);

(* ===== end of function ================================== *)

END_FUNCTION

